LIN {X 0,Y 92.351,Z 360.428,A -85,B 0,C 180,E1 -26835.446,E2 -26835.446} C_VEL
LIN {X 0,Y 91.502,Z 354.022,A -85,B 0,C 180,E1 -26842.823,E2 -26842.823} C_VEL
LIN {X 0,Y 91.802,Z 346.376,A -85,B 0,C 180,E1 -26849.841,E2 -26849.841} C_VEL
LIN {X 0,Y 92.482,Z 339.735,A -85,B 0,C 180,E1 -26854.849,E2 -26854.849} C_VEL
LIN {X 0,Y 93.803,Z 330.262,A -85,B 0,C 180,E1 -26860.681,E2 -26860.681} C_VEL
LIN {X 0,Y 95.598,Z 319.88,A -85,B 0,C 180,E1 -26865.787,E2 -26865.787} C_VEL
LIN {X 0,Y 97.517,Z 309.227,A -85,B 0,C 180,E1 -26869.896,E2 -26869.896} C_VEL
LIN {X 0,Y 99.765,Z 296.448,A -85,B 0,C 180,E1 -26873.677,E2 -26873.677} C_VEL
LIN {X 0,Y 101.625,Z 284.174,A -85,B 0,C 180,E1 -26876.408,E2 -26876.408} C_VEL
LIN {X 0,Y 103.341,Z 270.11,A -85,B 0,C 180,E1 -26878.615,E2 -26878.615} C_VEL
LIN {X 0,Y 107.967,Z 215.614,A -85,B 0,C 180,E1 -26883.951,E2 -26883.951} C_VEL
LIN {X 0,Y 101.224,Z 196.122,A -85,B 0,C 180,E1 -26887.415,E2 -26887.415} C_VEL
LIN {X 0,Y 94.785,Z 179.575,A -85,B 0,C 180,E1 -26890.931,E2 -26890.931} C_VEL
LIN {X 0,Y 93.797,Z 176.802,A -85,B 0,C 180,E1 -26891.572,E2 -26891.572} C_VEL
LIN {X 0,Y 94.063,Z 176.761,A -85,B 0,C 180,E1 -26897.046,E2 -26897.046} C_VEL
LIN {X 0,Y 94.193,Z 176.751,A -85,B 0,C 180,E1 -26901.416,E2 -26901.416} C_VEL
LIN {X 0,Y 94.794,Z 176.676,A -85,B 0,C 180,E1 -26909.998,E2 -26909.998} C_VEL
LIN {X 0,Y 94.198,Z 176.75,A -85,B 0,C 180,E1 -26918.58,E2 -26918.58} C_VEL
LIN {X 0,Y 94.04,Z 176.769,A -85,B 0,C 180,E1 -26923.708,E2 -26923.708} C_VEL
LIN {X 0,Y 93.691,Z 176.812,A -85,B 0,C 180,E1 -26932.027,E2 -26932.027} C_VEL
LIN {X 0,Y 93.619,Z 176.818,A -85,B 0,C 180,E1 -26936.769,E2 -26936.769} C_VEL
LIN {X 0,Y 93.61,Z 176.821,A -85,B 0,C 180,E1 -26944.328,E2 -26944.328} C_VEL
LIN {X 0,Y 93.63,Z 176.819,A -85,B 0,C 180,E1 -26952.495,E2 -26952.495} C_VEL
LIN {X 0,Y 93.626,Z 176.822,A -85,B 0,C 180,E1 -26958.644,E2 -26958.644} C_VEL
LIN {X 0,Y 93.611,Z 176.824,A -85,B 0,C 180,E1 -26965.671,E2 -26965.671} C_VEL
LIN {X 0,Y 93.666,Z 176.817,A -85,B 0,C 180,E1 -26974.205,E2 -26974.205} C_VEL
LIN {X 0,Y 93.691,Z 176.809,A -85,B 0,C 180,E1 -26977.974,E2 -26977.974} C_VEL
LIN {X 0,Y 94.089,Z 176.758,A -85,B 0,C 180,E1 -26987.053,E2 -26987.053} C_VEL
LIN {X 0,Y 94.198,Z 176.752,A -85,B 0,C 180,E1 -26991.42,E2 -26991.42} C_VEL
LIN {X 0,Y 94.794,Z 176.677,A -85,B 0,C 180,E1 -27000.002,E2 -27000.002} C_VEL
LIN {X 0,Y 94.21,Z 176.751,A -85,B 0,C 180,E1 -27008.582,E2 -27008.582} C_VEL
LIN {X 0,Y 94.034,Z 176.767,A -85,B 0,C 180,E1 -27013.693,E2 -27013.693} C_VEL
LIN {X 0,Y 93.692,Z 176.809,A -85,B 0,C 180,E1 -27022.03,E2 -27022.03} C_VEL
LIN {X 0,Y 93.62,Z 176.821,A -85,B 0,C 180,E1 -27026.772,E2 -27026.772} C_VEL
LIN {X 0,Y 93.599,Z 176.825,A -85,B 0,C 180,E1 -27034.318,E2 -27034.318} C_VEL
LIN {X 0,Y 93.641,Z 176.821,A -85,B 0,C 180,E1 -27042.076,E2 -27042.076} C_VEL
LIN {X 0,Y 94.743,Z 179.831,A -85,B 0,C 180,E1 -27042.784,E2 -27042.784} C_VEL
LIN {X 0,Y 98.916,Z 190.263,A -85,B 0,C 180,E1 -27045.097,E2 -27045.097} C_VEL
LIN {X 0,Y 105.331,Z 213.345,A -85,B 0,C 180,E1 -27049.033,E2 -27049.033} C_VEL
LIN {X 0,Y 106.725,Z 240.471,A -85,B 0,C 180,E1 -27052.191,E2 -27052.191} C_VEL
LIN {X 0,Y 103.42,Z 281.466,A -85,B 0,C 180,E1 -27056.341,E2 -27056.341} C_VEL
LIN {X 0,Y 101.758,Z 295.159,A -85,B 0,C 180,E1 -27058.514,E2 -27058.514} C_VEL
LIN {X 0,Y 99.924,Z 306.73,A -85,B 0,C 180,E1 -27061.085,E2 -27061.085} C_VEL
LIN {X 0,Y 97.629,Z 319.739,A -85,B 0,C 180,E1 -27064.982,E2 -27064.982} C_VEL
LIN {X 0,Y 95.507,Z 331.213,A -85,B 0,C 180,E1 -27069.543,E2 -27069.543} C_VEL
LIN {X 0,Y 94.096,Z 341.62,A -85,B 0,C 180,E1 -27074.848,E2 -27074.848} C_VEL
LIN {X 0,Y 93.264,Z 350.336,A -85,B 0,C 180,E1 -27080.438,E2 -27080.438} C_VEL
LIN {X 0,Y 93.204,Z 358.171,A -85,B 0,C 180,E1 -27086.76,E2 -27086.76} C_VEL
LIN {X 0,Y 93.403,Z 363.548,A -85,B 0,C 180,E1 -27092.158,E2 -27092.158} C_VEL
LIN {X 0,Y 92.94,Z 368.337,A -85,B 0,C 180,E1 -27098.7,E2 -27098.7} C_VEL
LIN {X 0,Y 93.452,Z 372.063,A -85,B 0,C 180,E1 -27105.263,E2 -27105.263} C_VEL
LIN {X 0,Y 95.199,Z 374.914,A -85,B 0,C 180,E1 -27111.663,E2 -27111.663} C_VEL
LIN {X 0,Y 99.586,Z 377.581,A -85,B 0,C 180,E1 -27119.606,E2 -27119.606} C_VEL
LIN {X 0,Y 106.025,Z 378.958,A -85,B 0,C 180,E1 -27126.627,E2 -27126.627} C_VEL
LIN {X 0,Y 114.018,Z 379.091,A -85,B 0,C 180,E1 -27132.692,E2 -27132.692} C_VEL
LIN {X 0,Y 123.472,Z 377.959,A -85,B 0,C 180,E1 -27137.729,E2 -27137.729} C_VEL
LIN {X 0,Y 134.03,Z 375.524,A -85,B 0,C 180,E1 -27141.865,E2 -27141.865} C_VEL
LIN {X 0,Y 145.317,Z 371.768,A -85,B 0,C 180,E1 -27145.305,E2 -27145.305} C_VEL
LIN {X 0,Y 154.3,Z 367.94,A -85,B 0,C 180,E1 -27147.421,E2 -27147.421} C_VEL
LIN {X 0,Y 160.353,Z 364.917,A -85,B 0,C 180,E1 -27148.639,E2 -27148.639} C_VEL
LIN {X 0,Y 160.723,Z 364.637,A -85,B 0,C 180,E1 -27149.394,E2 -27149.394} C_VEL
LIN {X 0,Y 149.736,Z 369.187,A -85,B 0,C 180,E1 -27152.006,E2 -27152.006} C_VEL
LIN {X 0,Y 139.588,Z 372.252,A -85,B 0,C 180,E1 -27154.996,E2 -27154.996} C_VEL
LIN {X 0,Y 137.751,Z 372.695,A -85,B 0,C 180,E1 -27155.614,E2 -27155.614} C_VEL
LIN {X 0,Y 132.899,Z 373.732,A -85,B 0,C 180,E1 -27156.983,E2 -27156.983} C_VEL
LIN {X 0,Y 123.979,Z 374.999,A -85,B 0,C 180,E1 -27158.851,E2 -27158.851} C_VEL
LIN {X 0,Y 115.232,Z 375.421,A -85,B 0,C 180,E1 -27161.053,E2 -27161.053} C_VEL
LIN {X 0,Y 110.768,Z 375.21,A -85,B 0,C 180,E1 -27162.998,E2 -27162.998} C_VEL
LIN {X 0,Y 103.035,Z 373.937,A -85,B 0,C 180,E1 -27168.191,E2 -27168.191} C_VEL
LIN {X 0,Y 98.79,Z 372.63,A -85,B 0,C 180,E1 -27171.819,E2 -27171.819} C_VEL
LIN {X 0,Y 93.327,Z 369.871,A -85,B 0,C 180,E1 -27177.841,E2 -27177.841} C_VEL
LIN {X 0,Y 89.087,Z 366.169,A -85,B 0,C 180,E1 -27184.523,E2 -27184.523} C_VEL
LIN {X 0,Y 86.188,Z 361.281,A -85,B 0,C 180,E1 -27191.892,E2 -27191.892} C_VEL
LIN {X 0,Y 84.732,Z 355.371,A -85,B 0,C 180,E1 -27199.375,E2 -27199.375} C_VEL
LIN {X 0,Y 84.582,Z 349.274,A -85,B 0,C 180,E1 -27205.861,E2 -27205.861} C_VEL
LIN {X 0,Y 85.129,Z 342.003,A -85,B 0,C 180,E1 -27212.225,E2 -27212.225} C_VEL
LIN {X 0,Y 86.35,Z 332.15,A -85,B 0,C 180,E1 -27219.105,E2 -27219.105} C_VEL
LIN {X 0,Y 88.2,Z 321.243,A -85,B 0,C 180,E1 -27225.064,E2 -27225.064} C_VEL
LIN {X 0,Y 90.086,Z 310.909,A -85,B 0,C 180,E1 -27229.518,E2 -27229.518} C_VEL
LIN {X 0,Y 92.208,Z 299.417,A -85,B 0,C 180,E1 -27233.381,E2 -27233.381} C_VEL
LIN {X 0,Y 94.384,Z 285.776,A -85,B 0,C 180,E1 -27236.815,E2 -27236.815} C_VEL
LIN {X 0,Y 96.163,Z 272.766,A -85,B 0,C 180,E1 -27239.129,E2 -27239.129} C_VEL
LIN {X 0,Y 98.117,Z 251.11,A -85,B 0,C 180,E1 -27241.602,E2 -27241.602} C_VEL
LIN {X 0,Y 101.067,Z 216.668,A -85,B 0,C 180,E1 -27245.079,E2 -27245.079} C_VEL
LIN {X 0,Y 93.632,Z 195.122,A -85,B 0,C 180,E1 -27249.255,E2 -27249.255} C_VEL
LIN {X 0,Y 87.72,Z 180.438,A -85,B 0,C 180,E1 -27252.769,E2 -27252.769} C_VEL
LIN {X 0,Y 86.787,Z 177.673,A -85,B 0,C 180,E1 -27253.533,E2 -27253.533} C_VEL
LIN {X 0,Y 87.097,Z 177.636,A -85,B 0,C 180,E1 -27260.711,E2 -27260.711} C_VEL
LIN {X 0,Y 87.721,Z 177.557,A -85,B 0,C 180,E1 -27269.998,E2 -27269.998} C_VEL
LIN {X 0,Y 87.106,Z 177.632,A -85,B 0,C 180,E1 -27279.284,E2 -27279.284} C_VEL
LIN {X 0,Y 86.948,Z 177.653,A -85,B 0,C 180,E1 -27284.086,E2 -27284.086} C_VEL
LIN {X 0,Y 86.584,Z 177.7,A -85,B 0,C 180,E1 -27293.942,E2 -27293.942} C_VEL
LIN {X 0,Y 86.475,Z 177.709,A -85,B 0,C 180,E1 -27299.183,E2 -27299.183} C_VEL
LIN {X 0,Y 86.535,Z 177.699,A -85,B 0,C 180,E1 -27305.695,E2 -27305.695} C_VEL
LIN {X 0,Y 86.557,Z 177.698,A -85,B 0,C 180,E1 -27313.053,E2 -27313.053} C_VEL
LIN {X 0,Y 86.55,Z 177.704,A -85,B 0,C 180,E1 -27319.49,E2 -27319.49} C_VEL
LIN {X 0,Y 86.559,Z 177.701,A -85,B 0,C 180,E1 -27325.367,E2 -27325.367} C_VEL
LIN {X 0,Y 86.583,Z 177.697,A -85,B 0,C 180,E1 -27333.233,E2 -27333.233} C_VEL
LIN {X 0,Y 86.645,Z 177.688,A -85,B 0,C 180,E1 -27341.07,E2 -27341.07} C_VEL
LIN {X 0,Y 86.967,Z 177.648,A -85,B 0,C 180,E1 -27345.971,E2 -27345.971} C_VEL
LIN {X 0,Y 87.106,Z 177.634,A -85,B 0,C 180,E1 -27350.716,E2 -27350.716} C_VEL
LIN {X 0,Y 87.721,Z 177.558,A -85,B 0,C 180,E1 -27360.002,E2 -27360.002} C_VEL
LIN {X 0,Y 87.114,Z 177.633,A -85,B 0,C 180,E1 -27369.287,E2 -27369.287} C_VEL
LIN {X 0,Y 86.949,Z 177.65,A -85,B 0,C 180,E1 -27374.089,E2 -27374.089} C_VEL
LIN {X 0,Y 86.586,Z 177.699,A -85,B 0,C 180,E1 -27383.946,E2 -27383.946} C_VEL
LIN {X 0,Y 86.475,Z 177.705,A -85,B 0,C 180,E1 -27389.187,E2 -27389.187} C_VEL
LIN {X 0,Y 86.521,Z 177.703,A -85,B 0,C 180,E1 -27395.683,E2 -27395.683} C_VEL
LIN {X 0,Y 86.529,Z 177.852,A -85,B 0,C 180,E1 -27400.186,E2 -27400.186} C_VEL
LIN {X 0,Y 88.646,Z 183.012,A -85,B 0,C 180,E1 -27401.528,E2 -27401.528} C_VEL
LIN {X 0,Y 92.717,Z 193.174,A -85,B 0,C 180,E1 -27403.954,E2 -27403.954} C_VEL
LIN {X 0,Y 98.684,Z 215.03,A -85,B 0,C 180,E1 -27407.971,E2 -27407.971} C_VEL
LIN {X 0,Y 99.874,Z 240.558,A -85,B 0,C 180,E1 -27411.166,E2 -27411.166} C_VEL
LIN {X 0,Y 96.441,Z 281.612,A -85,B 0,C 180,E1 -27415.616,E2 -27415.616} C_VEL
LIN {X 0,Y 94.812,Z 294.504,A -85,B 0,C 180,E1 -27417.808,E2 -27417.808} C_VEL
LIN {X 0,Y 92.919,Z 306.132,A -85,B 0,C 180,E1 -27420.554,E2 -27420.554} C_VEL
LIN {X 0,Y 90.555,Z 319.15,A -85,B 0,C 180,E1 -27424.734,E2 -27424.734} C_VEL
LIN {X 0,Y 88.426,Z 330.571,A -85,B 0,C 180,E1 -27429.654,E2 -27429.654} C_VEL
LIN {X 0,Y 87.135,Z 340.166,A -85,B 0,C 180,E1 -27434.926,E2 -27434.926} C_VEL
LIN {X 0,Y 86.384,Z 348.549,A -85,B 0,C 180,E1 -27440.637,E2 -27440.637} C_VEL
LIN {X 0,Y 86.382,Z 356.895,A -85,B 0,C 180,E1 -27447.67,E2 -27447.67} C_VEL
LIN {X 0,Y 86.603,Z 361.336,A -85,B 0,C 180,E1 -27452.327,E2 -27452.327} C_VEL
LIN {X 0,Y 86.258,Z 364.886,A -85,B 0,C 180,E1 -27457.022,E2 -27457.022} C_VEL
LIN {X 0,Y 86.463,Z 369.143,A -85,B 0,C 180,E1 -27464.116,E2 -27464.116} C_VEL
LIN {X 0,Y 88.757,Z 373.493,A -85,B 0,C 180,E1 -27473.325,E2 -27473.325} C_VEL
LIN {X 0,Y 93.53,Z 376.466,A -85,B 0,C 180,E1 -27481.737,E2 -27481.737} C_VEL
LIN {X 0,Y 100.426,Z 378.161,A -85,B 0,C 180,E1 -27489.04,E2 -27489.04} C_VEL
LIN {X 0,Y 108.92,Z 378.615,A -85,B 0,C 180,E1 -27495.218,E2 -27495.218} C_VEL
LIN {X 0,Y 118.822,Z 377.86,A -85,B 0,C 180,E1 -27500.258,E2 -27500.258} C_VEL
LIN {X 0,Y 129.784,Z 375.856,A -85,B 0,C 180,E1 -27504.32,E2 -27504.32} C_VEL
LIN {X 0,Y 141.416,Z 372.548,A -85,B 0,C 180,E1 -27507.658,E2 -27507.658} C_VEL
LIN {X 0,Y 147.52,Z 370.327,A -85,B 0,C 180,E1 -27509.043,E2 -27509.043} C_VEL
LIN {X 0,Y 146.705,Z 370.553,A -85,B 0,C 180,E1 -27509.578,E2 -27509.578} C_VEL
LIN {X 0,Y 133.944,Z 373.781,A -85,B 0,C 180,E1 -27513.126,E2 -27513.126} C_VEL
LIN {X 0,Y 121.594,Z 375.353,A -85,B 0,C 180,E1 -27517.638,E2 -27517.638} C_VEL
LIN {X 0,Y 110.768,Z 375.21,A -85,B 0,C 180,E1 -27522.998,E2 -27522.998} C_VEL
LIN {X 0,Y 106.467,Z 374.769,A -85,B 0,C 180,E1 -27525.123,E2 -27525.123} C_VEL
LIN {X 0,Y 98.494,Z 373.407,A -85,B 0,C 180,E1 -27528.331,E2 -27528.331} C_VEL
LIN {X 0,Y 91.021,Z 371.275,A -85,B 0,C 180,E1 -27532.057,E2 -27532.057} C_VEL
LIN {X 0,Y 87.655,Z 369.634,A -85,B 0,C 180,E1 -27535.004,E2 -27535.004} C_VEL
LIN {X 0,Y 82.729,Z 365.476,A -85,B 0,C 180,E1 -27542.433,E2 -27542.433} C_VEL
LIN {X 0,Y 79.044,Z 359.168,A -85,B 0,C 180,E1 -27552.021,E2 -27552.021} C_VEL
LIN {X 0,Y 77.691,Z 351.807,A -85,B 0,C 180,E1 -27561.212,E2 -27561.212} C_VEL
LIN {X 0,Y 77.776,Z 344.892,A -85,B 0,C 180,E1 -27568.318,E2 -27568.318} C_VEL
LIN {X 0,Y 78.474,Z 337.481,A -85,B 0,C 180,E1 -27574.618,E2 -27574.618} C_VEL
LIN {X 0,Y 79.851,Z 327.7,A -85,B 0,C 180,E1 -27581.305,E2 -27581.305} C_VEL
LIN {X 0,Y 81.805,Z 316.889,A -85,B 0,C 180,E1 -27587.09,E2 -27587.09} C_VEL
LIN {X 0,Y 83.908,Z 305.754,A -85,B 0,C 180,E1 -27591.74,E2 -27591.74} C_VEL
LIN {X 0,Y 86.18,Z 293.338,A -85,B 0,C 180,E1 -27595.656,E2 -27595.656} C_VEL
LIN {X 0,Y 88.299,Z 279.63,A -85,B 0,C 180,E1 -27598.825,E2 -27598.825} C_VEL
LIN {X 0,Y 89.719,Z 267.085,A -85,B 0,C 180,E1 -27600.824,E2 -27600.824} C_VEL
LIN {X 0,Y 94.234,Z 217.928,A -85,B 0,C 180,E1 -27606.271,E2 -27606.271} C_VEL
LIN {X 0,Y 87.202,Z 197.474,A -85,B 0,C 180,E1 -27610.578,E2 -27610.578} C_VEL
LIN {X 0,Y 81.948,Z 184.113,A -85,B 0,C 180,E1 -27614.054,E2 -27614.054} C_VEL
LIN {X 0,Y 79.877,Z 178.778,A -85,B 0,C 180,E1 -27615.579,E2 -27615.579} C_VEL
LIN {X 0,Y 79.865,Z 178.529,A -85,B 0,C 180,E1 -27615.871,E2 -27615.871} C_VEL
LIN {X 0,Y 79.976,Z 178.523,A -85,B 0,C 180,E1 -27619.876,E2 -27619.876} C_VEL
LIN {X 0,Y 80.649,Z 178.439,A -85,B 0,C 180,E1 -27629.998,E2 -27629.998} C_VEL
LIN {X 0,Y 79.991,Z 178.515,A -85,B 0,C 180,E1 -27640.119,E2 -27640.119} C_VEL
LIN {X 0,Y 79.76,Z 178.55,A -85,B 0,C 180,E1 -27645.326,E2 -27645.326} C_VEL
LIN {X 0,Y 79.511,Z 178.574,A -85,B 0,C 180,E1 -27650.703,E2 -27650.703} C_VEL
LIN {X 0,Y 79.48,Z 178.577,A -85,B 0,C 180,E1 -27657.845,E2 -27657.845} C_VEL
LIN {X 0,Y 79.449,Z 178.583,A -85,B 0,C 180,E1 -27667.241,E2 -27667.241} C_VEL
LIN {X 0,Y 79.464,Z 178.579,A -85,B 0,C 180,E1 -27675.032,E2 -27675.032} C_VEL
LIN {X 0,Y 79.45,Z 178.58,A -85,B 0,C 180,E1 -27682.758,E2 -27682.758} C_VEL
LIN {X 0,Y 79.482,Z 178.579,A -85,B 0,C 180,E1 -27692.153,E2 -27692.153} C_VEL
LIN {X 0,Y 79.512,Z 178.573,A -85,B 0,C 180,E1 -27699.297,E2 -27699.297} C_VEL
LIN {X 0,Y 79.839,Z 178.537,A -85,B 0,C 180,E1 -27705.527,E2 -27705.527} C_VEL
LIN {X 0,Y 79.991,Z 178.519,A -85,B 0,C 180,E1 -27709.881,E2 -27709.881} C_VEL
LIN {X 0,Y 80.649,Z 178.439,A -85,B 0,C 180,E1 -27720.002,E2 -27720.002} C_VEL
LIN {X 0,Y 79.993,Z 178.518,A -85,B 0,C 180,E1 -27730.122,E2 -27730.122} C_VEL
LIN {X 0,Y 79.761,Z 178.549,A -85,B 0,C 180,E1 -27735.33,E2 -27735.33} C_VEL
LIN {X 0,Y 79.513,Z 178.573,A -85,B 0,C 180,E1 -27740.707,E2 -27740.707} C_VEL
LIN {X 0,Y 79.481,Z 178.578,A -85,B 0,C 180,E1 -27747.847,E2 -27747.847} C_VEL
LIN {X 0,Y 79.443,Z 178.581,A -85,B 0,C 180,E1 -27757.235,E2 -27757.235} C_VEL
LIN {X 0,Y 79.44,Z 178.582,A -85,B 0,C 180,E1 -27757.878,E2 -27757.878} C_VEL
LIN {X 0,Y 80.432,Z 181.432,A -85,B 0,C 180,E1 -27758.708,E2 -27758.708} C_VEL
LIN {X 0,Y 85.393,Z 192.723,A -85,B 0,C 180,E1 -27761.942,E2 -27761.942} C_VEL
LIN {X 0,Y 89.063,Z 205.266,A -85,B 0,C 180,E1 -27764.626,E2 -27764.626} C_VEL
LIN {X 0,Y 92.048,Z 217.164,A -85,B 0,C 180,E1 -27766.835,E2 -27766.835} C_VEL
LIN {X 0,Y 93.078,Z 240.438,A -85,B 0,C 180,E1 -27769.967,E2 -27769.967} C_VEL
LIN {X 0,Y 89.562,Z 280.628,A -85,B 0,C 180,E1 -27774.641,E2 -27774.641} C_VEL
LIN {X 0,Y 87.906,Z 293.587,A -85,B 0,C 180,E1 -27777.001,E2 -27777.001} C_VEL
LIN {X 0,Y 85.956,Z 305.243,A -85,B 0,C 180,E1 -27779.949,E2 -27779.949} C_VEL
LIN {X 0,Y 83.546,Z 318.246,A -85,B 0,C 180,E1 -27784.463,E2 -27784.463} C_VEL
LIN {X 0,Y 81.385,Z 329.761,A -85,B 0,C 180,E1 -27789.795,E2 -27789.795} C_VEL
LIN {X 0,Y 79.98,Z 340.754,A -85,B 0,C 180,E1 -27796.433,E2 -27796.433} C_VEL
LIN {X 0,Y 79.417,Z 348.596,A -85,B 0,C 180,E1 -27802.374,E2 -27802.374} C_VEL
LIN {X 0,Y 79.585,Z 355.553,A -85,B 0,C 180,E1 -27808.737,E2 -27808.737} C_VEL
LIN {X 0,Y 79.808,Z 359.014,A -85,B 0,C 180,E1 -27812.525,E2 -27812.525} C_VEL
LIN {X 0,Y 79.568,Z 362.74,A -85,B 0,C 180,E1 -27817.615,E2 -27817.615} C_VEL
LIN {X 0,Y 80.239,Z 368.574,A -85,B 0,C 180,E1 -27827.854,E2 -27827.854} C_VEL
LIN {X 0,Y 82.417,Z 371.927,A -85,B 0,C 180,E1 -27835.239,E2 -27835.239} C_VEL
LIN {X 0,Y 87.664,Z 375.208,A -85,B 0,C 180,E1 -27844.14,E2 -27844.14} C_VEL
LIN {X 0,Y 95.053,Z 377.24,A -85,B 0,C 180,E1 -27851.718,E2 -27851.718} C_VEL
LIN {X 0,Y 104.064,Z 378.056,A -85,B 0,C 180,E1 -27857.98,E2 -27857.98} C_VEL
LIN {X 0,Y 114.428,Z 377.687,A -85,B 0,C 180,E1 -27862.984,E2 -27862.984} C_VEL
LIN {X 0,Y 125.782,Z 376.089,A -85,B 0,C 180,E1 -27866.944,E2 -27866.944} C_VEL
LIN {X 0,Y 131.672,Z 374.799,A -85,B 0,C 180,E1 -27868.651,E2 -27868.651} C_VEL
LIN {X 0,Y 133.177,Z 374.323,A -85,B 0,C 180,E1 -27869.701,E2 -27869.701} C_VEL
LIN {X 0,Y 123.077,Z 375.674,A -85,B 0,C 180,E1 -27872.817,E2 -27872.817} C_VEL
LIN {X 0,Y 115.793,Z 376.028,A -85,B 0,C 180,E1 -27875.567,E2 -27875.567} C_VEL
LIN {X 0,Y 105.417,Z 375.414,A -85,B 0,C 180,E1 -27880.527,E2 -27880.527} C_VEL
LIN {X 0,Y 95.489,Z 373.242,A -85,B 0,C 180,E1 -27887.242,E2 -27887.242} C_VEL
LIN {X 0,Y 89.18,Z 370.55,A -85,B 0,C 180,E1 -27893.209,E2 -27893.209} C_VEL
LIN {X 0,Y 87.655,Z 369.634,A -85,B 0,C 180,E1 -27895.004,E2 -27895.004} C_VEL
LIN {X 0,Y 84.598,Z 367.791,A -85,B 0,C 180,E1 -27898.135,E2 -27898.135} C_VEL
LIN {X 0,Y 78.699,Z 364.017,A -85,B 0,C 180,E1 -27903.064,E2 -27903.064} C_VEL
LIN {X 0,Y 73.582,Z 359.497,A -85,B 0,C 180,E1 -27908.531,E2 -27908.531} C_VEL
LIN {X 0,Y 71.904,Z 356.563,A -85,B 0,C 180,E1 -27912.38,E2 -27912.38} C_VEL
LIN {X 0,Y 70.76,Z 349.115,A -85,B 0,C 180,E1 -27921.865,E2 -27921.865} C_VEL
LIN {X 0,Y 71.017,Z 341.606,A -85,B 0,C 180,E1 -27929.655,E2 -27929.655} C_VEL
LIN {X 0,Y 71.958,Z 332.755,A -85,B 0,C 180,E1 -27937.081,E2 -27937.081} C_VEL
LIN {X 0,Y 73.55,Z 322.642,A -85,B 0,C 180,E1 -27943.847,E2 -27943.847} C_VEL
LIN {X 0,Y 75.73,Z 311.186,A -85,B 0,C 180,E1 -27949.834,E2 -27949.834} C_VEL
LIN {X 0,Y 77.906,Z 299.975,A -85,B 0,C 180,E1 -27954.278,E2 -27954.278} C_VEL
LIN {X 0,Y 80.336,Z 286.072,A -85,B 0,C 180,E1 -27958.336,E2 -27958.336} C_VEL
LIN {X 0,Y 82.359,Z 271.903,A -85,B 0,C 180,E1 -27961.16,E2 -27961.16} C_VEL
LIN {X 0,Y 86.345,Z 230.389,A -85,B 0,C 180,E1 -27966.296,E2 -27966.296} C_VEL
LIN {X 0,Y 87.453,Z 219.393,A -85,B 0,C 180,E1 -27967.533,E2 -27967.533} C_VEL
LIN {X 0,Y 81.166,Z 200.697,A -85,B 0,C 180,E1 -27971.868,E2 -27971.868} C_VEL
LIN {X 0,Y 76.043,Z 187.435,A -85,B 0,C 180,E1 -27975.606,E2 -27975.606} C_VEL
LIN {X 0,Y 72.922,Z 179.748,A -85,B 0,C 180,E1 -27978.112,E2 -27978.112} C_VEL
LIN {X 0,Y 72.865,Z 179.406,A -85,B 0,C 180,E1 -27978.489,E2 -27978.489} C_VEL
LIN {X 0,Y 73.575,Z 179.32,A -85,B 0,C 180,E1 -27989.998,E2 -27989.998} C_VEL
LIN {X 0,Y 72.878,Z 179.399,A -85,B 0,C 180,E1 -28001.118,E2 -28001.118} C_VEL
LIN {X 0,Y 72.58,Z 179.443,A -85,B 0,C 180,E1 -28006.885,E2 -28006.885} C_VEL
LIN {X 0,Y 72.391,Z 179.468,A -85,B 0,C 180,E1 -28012.849,E2 -28012.849} C_VEL
LIN {X 0,Y 72.373,Z 179.464,A -85,B 0,C 180,E1 -28019.081,E2 -28019.081} C_VEL
LIN {X 0,Y 72.335,Z 179.467,A -85,B 0,C 180,E1 -28025.656,E2 -28025.656} C_VEL
LIN {X 0,Y 72.31,Z 179.473,A -85,B 0,C 180,E1 -28032.868,E2 -28032.868} C_VEL
LIN {X 0,Y 72.357,Z 179.467,A -85,B 0,C 180,E1 -28040.987,E2 -28040.987} C_VEL
LIN {X 0,Y 72.336,Z 179.47,A -85,B 0,C 180,E1 -28044.344,E2 -28044.344} C_VEL
LIN {X 0,Y 72.389,Z 179.46,A -85,B 0,C 180,E1 -28050.961,E2 -28050.961} C_VEL
LIN {X 0,Y 72.392,Z 179.464,A -85,B 0,C 180,E1 -28057.152,E2 -28057.152} C_VEL
LIN {X 0,Y 72.733,Z 179.423,A -85,B 0,C 180,E1 -28065.068,E2 -28065.068} C_VEL
LIN {X 0,Y 72.878,Z 179.401,A -85,B 0,C 180,E1 -28068.882,E2 -28068.882} C_VEL
LIN {X 0,Y 73.575,Z 179.32,A -85,B 0,C 180,E1 -28080.002,E2 -28080.002} C_VEL
LIN {X 0,Y 72.878,Z 179.401,A -85,B 0,C 180,E1 -28091.122,E2 -28091.122} C_VEL
LIN {X 0,Y 72.581,Z 179.444,A -85,B 0,C 180,E1 -28096.889,E2 -28096.889} C_VEL
LIN {X 0,Y 72.393,Z 179.464,A -85,B 0,C 180,E1 -28102.853,E2 -28102.853} C_VEL
LIN {X 0,Y 72.376,Z 179.461,A -85,B 0,C 180,E1 -28109.085,E2 -28109.085} C_VEL
LIN {X 0,Y 72.306,Z 179.475,A -85,B 0,C 180,E1 -28115.25,E2 -28115.25} C_VEL
LIN {X 0,Y 73.4,Z 182.395,A -85,B 0,C 180,E1 -28116.217,E2 -28116.217} C_VEL
LIN {X 0,Y 78.274,Z 193.22,A -85,B 0,C 180,E1 -28119.774,E2 -28119.774} C_VEL
LIN {X 0,Y 80.557,Z 199.631,A -85,B 0,C 180,E1 -28121.493,E2 -28121.493} C_VEL
LIN {X 0,Y 85.327,Z 218.12,A -85,B 0,C 180,E1 -28125.462,E2 -28125.462} C_VEL
LIN {X 0,Y 86.228,Z 240.55,A -85,B 0,C 180,E1 -28128.73,E2 -28128.73} C_VEL
LIN {X 0,Y 82.567,Z 280.829,A -85,B 0,C 180,E1 -28133.809,E2 -28133.809} C_VEL
LIN {X 0,Y 80.846,Z 293.597,A -85,B 0,C 180,E1 -28136.348,E2 -28136.348} C_VEL
LIN {X 0,Y 78.654,Z 305.996,A -85,B 0,C 180,E1 -28139.829,E2 -28139.829} C_VEL
LIN {X 0,Y 76.542,Z 317.338,A -85,B 0,C 180,E1 -28144.144,E2 -28144.144} C_VEL
LIN {X 0,Y 74.337,Z 328.947,A -85,B 0,C 180,E1 -28149.962,E2 -28149.962} C_VEL
LIN {X 0,Y 73.023,Z 339.669,A -85,B 0,C 180,E1 -28157.015,E2 -28157.015} C_VEL
LIN {X 0,Y 72.564,Z 348.536,A -85,B 0,C 180,E1 -28164.444,E2 -28164.444} C_VEL
LIN {X 0,Y 72.962,Z 355.297,A -85,B 0,C 180,E1 -28171.382,E2 -28171.382} C_VEL
LIN {X 0,Y 73.103,Z 358.606,A -85,B 0,C 180,E1 -28175.519,E2 -28175.519} C_VEL
LIN {X 0,Y 72.934,Z 363.505,A -85,B 0,C 180,E1 -28183.459,E2 -28183.459} C_VEL
LIN {X 0,Y 74.405,Z 367.92,A -85,B 0,C 180,E1 -28192.201,E2 -28192.201} C_VEL
LIN {X 0,Y 78.79,Z 372.206,A -85,B 0,C 180,E1 -28202.359,E2 -28202.359} C_VEL
LIN {X 0,Y 85.711,Z 375.195,A -85,B 0,C 180,E1 -28210.996,E2 -28210.996} C_VEL
LIN {X 0,Y 94.509,Z 376.966,A -85,B 0,C 180,E1 -28218.044,E2 -28218.044} C_VEL
LIN {X 0,Y 104.738,Z 377.54,A -85,B 0,C 180,E1 -28223.633,E2 -28223.633} C_VEL
LIN {X 0,Y 116.085,Z 376.929,A -85,B 0,C 180,E1 -28227.953,E2 -28227.953} C_VEL
LIN {X 0,Y 118.009,Z 376.707,A -85,B 0,C 180,E1 -28228.548,E2 -28228.548} C_VEL
LIN {X 0,Y 119.865,Z 376.399,A -85,B 0,C 180,E1 -28229.828,E2 -28229.828} C_VEL
LIN {X 0,Y 109.849,Z 376.469,A -85,B 0,C 180,E1 -28233.393,E2 -28233.393} C_VEL
LIN {X 0,Y 98.131,Z 375.095,A -85,B 0,C 180,E1 -28239.015,E2 -28239.015} C_VEL
LIN {X 0,Y 87.951,Z 372.179,A -85,B 0,C 180,E1 -28246.128,E2 -28246.128} C_VEL
LIN {X 0,Y 79.723,Z 367.624,A -85,B 0,C 180,E1 -28254.941,E2 -28254.941} C_VEL
LIN {X 0,Y 75.173,Z 363.052,A -85,B 0,C 180,E1 -28262.677,E2 -28262.677} C_VEL
LIN {X 0,Y 71.904,Z 356.563,A -85,B 0,C 180,E1 -28272.38,E2 -28272.38} C_VEL
LIN {X 0,Y 70.592,Z 353.473,A -85,B 0,C 180,E1 -28276.255,E2 -28276.255} C_VEL
LIN {X 0,Y 68.718,Z 350.021,A -85,B 0,C 180,E1 -28279.92,E2 -28279.92} C_VEL
LIN {X 0,Y 65.106,Z 342.359,A -85,B 0,C 180,E1 -28287.233,E2 -28287.233} C_VEL
LIN {X 0,Y 64.351,Z 338.253,A -85,B 0,C 180,E1 -28291.038,E2 -28291.038} C_VEL
LIN {X 0,Y 64.387,Z 336.838,A -85,B 0,C 180,E1 -28292.312,E2 -28292.312} C_VEL
LIN {X 0,Y 65.744,Z 326.301,A -85,B 0,C 180,E1 -28300.873,E2 -28300.873} C_VEL
LIN {X 0,Y 67.713,Z 315.47,A -85,B 0,C 180,E1 -28307.686,E2 -28307.686} C_VEL
LIN {X 0,Y 70.05,Z 303.585,A -85,B 0,C 180,E1 -28313.378,E2 -28313.378} C_VEL
LIN {X 0,Y 72.322,Z 291.896,A -85,B 0,C 180,E1 -28317.585,E2 -28317.585} C_VEL
LIN {X 0,Y 74.66,Z 277.702,A -85,B 0,C 180,E1 -28321.212,E2 -28321.212} C_VEL
LIN {X 0,Y 76.261,Z 263.956,A -85,B 0,C 180,E1 -28323.566,E2 -28323.566} C_VEL
LIN {X 0,Y 80.665,Z 220.64,A -85,B 0,C 180,E1 -28329.06,E2 -28329.06} C_VEL
LIN {X 0,Y 74.815,Z 203.089,A -85,B 0,C 180,E1 -28333.495,E2 -28333.495} C_VEL
LIN {X 0,Y 70.277,Z 190.976,A -85,B 0,C 180,E1 -28337.255,E2 -28337.255} C_VEL
LIN {X 0,Y 66.729,Z 182.984,A -85,B 0,C 180,E1 -28340.335,E2 -28340.335} C_VEL
LIN {X 0,Y 65.823,Z 180.285,A -85,B 0,C 180,E1 -28341.362,E2 -28341.362} C_VEL
LIN {X 0,Y 66.499,Z 180.201,A -85,B 0,C 180,E1 -28349.998,E2 -28349.998} C_VEL
LIN {X 0,Y 65.77,Z 180.285,A -85,B 0,C 180,E1 -28362.338,E2 -28362.338} C_VEL
LIN {X 0,Y 65.382,Z 180.333,A -85,B 0,C 180,E1 -28368.81,E2 -28368.81} C_VEL
LIN {X 0,Y 65.243,Z 180.355,A -85,B 0,C 180,E1 -28375.521,E2 -28375.521} C_VEL
LIN {X 0,Y 65.212,Z 180.362,A -85,B 0,C 180,E1 -28382.603,E2 -28382.603} C_VEL
LIN {X 0,Y 65.247,Z 180.357,A -85,B 0,C 180,E1 -28391.066,E2 -28391.066} C_VEL
LIN {X 0,Y 65.264,Z 180.354,A -85,B 0,C 180,E1 -28399.754,E2 -28399.754} C_VEL
LIN {X 0,Y 65.257,Z 180.351,A -85,B 0,C 180,E1 -28409.49,E2 -28409.49} C_VEL
LIN {X 0,Y 65.245,Z 180.358,A -85,B 0,C 180,E1 -28414.48,E2 -28414.48} C_VEL
LIN {X 0,Y 65.634,Z 180.309,A -85,B 0,C 180,E1 -28424.509,E2 -28424.509} C_VEL
LIN {X 0,Y 65.77,Z 180.284,A -85,B 0,C 180,E1 -28427.662,E2 -28427.662} C_VEL
LIN {X 0,Y 66.499,Z 180.202,A -85,B 0,C 180,E1 -28440.002,E2 -28440.002} C_VEL
LIN {X 0,Y 65.778,Z 180.283,A -85,B 0,C 180,E1 -28452.341,E2 -28452.341} C_VEL
LIN {X 0,Y 65.384,Z 180.336,A -85,B 0,C 180,E1 -28458.814,E2 -28458.814} C_VEL
LIN {X 0,Y 65.238,Z 180.359,A -85,B 0,C 180,E1 -28465.528,E2 -28465.528} C_VEL
LIN {X 0,Y 65.292,Z 180.351,A -85,B 0,C 180,E1 -28472.075,E2 -28472.075} C_VEL
LIN {X 0,Y 66.418,Z 183.431,A -85,B 0,C 180,E1 -28473.294,E2 -28473.294} C_VEL
LIN {X 0,Y 71.516,Z 194.42,A -85,B 0,C 180,E1 -28477.531,E2 -28477.531} C_VEL
LIN {X 0,Y 74.266,Z 201.919,A -85,B 0,C 180,E1 -28479.782,E2 -28479.782} C_VEL
LIN {X 0,Y 78.68,Z 219.568,A -85,B 0,C 180,E1 -28483.934,E2 -28483.934} C_VEL
LIN {X 0,Y 79.422,Z 240.914,A -85,B 0,C 180,E1 -28487.336,E2 -28487.336} C_VEL
LIN {X 0,Y 75.676,Z 280.153,A -85,B 0,C 180,E1 -28492.662,E2 -28492.662} C_VEL
LIN {X 0,Y 73.801,Z 293.612,A -85,B 0,C 180,E1 -28495.571,E2 -28495.571} C_VEL
LIN {X 0,Y 71.37,Z 306.72,A -85,B 0,C 180,E1 -28499.693,E2 -28499.693} C_VEL
LIN {X 0,Y 69.247,Z 317.733,A -85,B 0,C 180,E1 -28504.45,E2 -28504.45} C_VEL
LIN {X 0,Y 67.21,Z 328.731,A -85,B 0,C 180,E1 -28510.692,E2 -28510.692} C_VEL
LIN {X 0,Y 66.11,Z 338.381,A -85,B 0,C 180,E1 -28517.727,E2 -28517.727} C_VEL
LIN {X 0,Y 65.769,Z 346.84,A -85,B 0,C 180,E1 -28525.405,E2 -28525.405} C_VEL
LIN {X 0,Y 66.307,Z 353.782,A -85,B 0,C 180,E1 -28533.04,E2 -28533.04} C_VEL
LIN {X 0,Y 66.462,Z 356.104,A -85,B 0,C 180,E1 -28536.072,E2 -28536.072} C_VEL
LIN {X 0,Y 66.524,Z 361.868,A -85,B 0,C 180,E1 -28545.973,E2 -28545.973} C_VEL
LIN {X 0,Y 69.102,Z 367.227,A -85,B 0,C 180,E1 -28557.239,E2 -28557.239} C_VEL
LIN {X 0,Y 73.044,Z 370.577,A -85,B 0,C 180,E1 -28565.263,E2 -28565.263} C_VEL
LIN {X 0,Y 80.56,Z 373.874,A -85,B 0,C 180,E1 -28574.262,E2 -28574.262} C_VEL
LIN {X 0,Y 89.958,Z 375.97,A -85,B 0,C 180,E1 -28581.378,E2 -28581.378} C_VEL
LIN {X 0,Y 100.707,Z 376.905,A -85,B 0,C 180,E1 -28586.873,E2 -28586.873} C_VEL
LIN {X 0,Y 106.518,Z 376.949,A -85,B 0,C 180,E1 -28589.065,E2 -28589.065} C_VEL
LIN {X 0,Y 104.762,Z 376.712,A -85,B 0,C 180,E1 -28590.707,E2 -28590.707} C_VEL
LIN {X 0,Y 96.729,Z 375.645,A -85,B 0,C 180,E1 -28594.153,E2 -28594.153} C_VEL
LIN {X 0,Y 85.488,Z 372.78,A -85,B 0,C 180,E1 -28600.8,E2 -28600.8} C_VEL
LIN {X 0,Y 78.146,Z 369.508,A -85,B 0,C 180,E1 -28607.095,E2 -28607.095} C_VEL
LIN {X 0,Y 72.195,Z 365.399,A -85,B 0,C 180,E1 -28614.411,E2 -28614.411} C_VEL
LIN {X 0,Y 67.09,Z 359.292,A -85,B 0,C 180,E1 -28624.504,E2 -28624.504} C_VEL
LIN {X 0,Y 64.33,Z 351.422,A -85,B 0,C 180,E1 -28635.844,E2 -28635.844} C_VEL
LIN {X 0,Y 63.899,Z 344.564,A -85,B 0,C 180,E1 -28644.356,E2 -28644.356} C_VEL
LIN {X 0,Y 64.387,Z 336.838,A -85,B 0,C 180,E1 -28652.312,E2 -28652.312} C_VEL
LIN {X 0,Y 64.172,Z 332.601,A -85,B 0,C 180,E1 -28655.902,E2 -28655.902} C_VEL
LIN {X 0,Y 62.385,Z 324.99,A -85,B 0,C 180,E1 -28661.426,E2 -28661.426} C_VEL
LIN {X 0,Y 60.912,Z 316.862,A -85,B 0,C 180,E1 -28666.736,E2 -28666.736} C_VEL
LIN {X 0,Y 61.236,Z 311.795,A -85,B 0,C 180,E1 -28669.719,E2 -28669.719} C_VEL
LIN {X 0,Y 63.701,Z 299.814,A -85,B 0,C 180,E1 -28675.499,E2 -28675.499} C_VEL
LIN {X 0,Y 66.291,Z 286.285,A -85,B 0,C 180,E1 -28680.224,E2 -28680.224} C_VEL
LIN {X 0,Y 68.588,Z 271.36,A -85,B 0,C 180,E1 -28683.707,E2 -28683.707} C_VEL
LIN {X 0,Y 73.816,Z 221.568,A -85,B 0,C 180,E1 -28690.799,E2 -28690.799} C_VEL
LIN {X 0,Y 67.875,Z 203.568,A -85,B 0,C 180,E1 -28695.988,E2 -28695.988} C_VEL
LIN {X 0,Y 62.811,Z 190.132,A -85,B 0,C 180,E1 -28700.942,E2 -28700.942} C_VEL
LIN {X 0,Y 59.071,Z 181.858,A -85,B 0,C 180,E1 -28704.878,E2 -28704.878} C_VEL
LIN {X 0,Y 58.954,Z 181.133,A -85,B 0,C 180,E1 -28705.296,E2 -28705.296} C_VEL
LIN {X 0,Y 59.39,Z 181.086,A -85,B 0,C 180,E1 -28709.997,E2 -28709.997} C_VEL
LIN {X 0,Y 58.816,Z 181.159,A -85,B 0,C 180,E1 -28716.86,E2 -28716.86} C_VEL
LIN {X 0,Y 58.523,Z 181.195,A -85,B 0,C 180,E1 -28726.122,E2 -28726.122} C_VEL
LIN {X 0,Y 58.153,Z 181.234,A -85,B 0,C 180,E1 -28738.906,E2 -28738.906} C_VEL
LIN {X 0,Y 58.072,Z 181.244,A -85,B 0,C 180,E1 -28747.234,E2 -28747.234} C_VEL
LIN {X 0,Y 58.092,Z 181.245,A -85,B 0,C 180,E1 -28756.539,E2 -28756.539} C_VEL
LIN {X 0,Y 58.072,Z 181.242,A -85,B 0,C 180,E1 -28762.766,E2 -28762.766} C_VEL
LIN {X 0,Y 58.153,Z 181.232,A -85,B 0,C 180,E1 -28771.095,E2 -28771.095} C_VEL
LIN {X 0,Y 58.523,Z 181.195,A -85,B 0,C 180,E1 -28783.878,E2 -28783.878} C_VEL
LIN {X 0,Y 58.815,Z 181.157,A -85,B 0,C 180,E1 -28793.14,E2 -28793.14} C_VEL
LIN {X 0,Y 59.391,Z 181.087,A -85,B 0,C 180,E1 -28800.003,E2 -28800.003} C_VEL
LIN {X 0,Y 58.821,Z 181.156,A -85,B 0,C 180,E1 -28806.865,E2 -28806.865} C_VEL
LIN {X 0,Y 58.655,Z 181.173,A -85,B 0,C 180,E1 -28813.868,E2 -28813.868} C_VEL
LIN {X 0,Y 58.163,Z 181.235,A -85,B 0,C 180,E1 -28826.947,E2 -28826.947} C_VEL
LIN {X 0,Y 58.161,Z 181.232,A -85,B 0,C 180,E1 -28827.923,E2 -28827.923} C_VEL
LIN {X 0,Y 59.245,Z 184.121,A -85,B 0,C 180,E1 -28829.386,E2 -28829.386} C_VEL
LIN {X 0,Y 60.654,Z 186.718,A -85,B 0,C 180,E1 -28830.831,E2 -28830.831} C_VEL
LIN {X 0,Y 65.006,Z 196.153,A -85,B 0,C 180,E1 -28835.057,E2 -28835.057} C_VEL
LIN {X 0,Y 68.001,Z 204.366,A -85,B 0,C 180,E1 -28837.901,E2 -28837.901} C_VEL
LIN {X 0,Y 72.026,Z 220.855,A -85,B 0,C 180,E1 -28842.177,E2 -28842.177} C_VEL
LIN {X 0,Y 72.638,Z 241.116,A -85,B 0,C 180,E1 -28845.69,E2 -28845.69} C_VEL
LIN {X 0,Y 68.753,Z 279.864,A -85,B 0,C 180,E1 -28851.474,E2 -28851.474} C_VEL
LIN {X 0,Y 66.817,Z 293.175,A -85,B 0,C 180,E1 -28854.658,E2 -28854.658} C_VEL
LIN {X 0,Y 64.479,Z 305.3,A -85,B 0,C 180,E1 -28858.823,E2 -28858.823} C_VEL
LIN {X 0,Y 62.176,Z 316.965,A -85,B 0,C 180,E1 -28864.337,E2 -28864.337} C_VEL
LIN {X 0,Y 60.264,Z 327.3,A -85,B 0,C 180,E1 -28870.794,E2 -28870.794} C_VEL
LIN {X 0,Y 59.26,Z 336.451,A -85,B 0,C 180,E1 -28878.024,E2 -28878.024} C_VEL
LIN {X 0,Y 59.003,Z 345.146,A -85,B 0,C 180,E1 -28886.588,E2 -28886.588} C_VEL
LIN {X 0,Y 59.735,Z 352.199,A -85,B 0,C 180,E1 -28895.065,E2 -28895.065} C_VEL
LIN {X 0,Y 59.831,Z 355.473,A -85,B 0,C 180,E1 -28900.151,E2 -28900.151} C_VEL
LIN {X 0,Y 60.914,Z 361.849,A -85,B 0,C 180,E1 -28912.625,E2 -28912.625} C_VEL
LIN {X 0,Y 64.391,Z 366.454,A -85,B 0,C 180,E1 -28923.077,E2 -28923.077} C_VEL
LIN {X 0,Y 71.366,Z 370.741,A -85,B 0,C 180,E1 -28933.582,E2 -28933.582} C_VEL
LIN {X 0,Y 80.573,Z 373.785,A -85,B 0,C 180,E1 -28941.726,E2 -28941.726} C_VEL
LIN {X 0,Y 92.634,Z 375.823,A -85,B 0,C 180,E1 -28948.534,E2 -28948.534} C_VEL
LIN {X 0,Y 93.938,Z 375.834,A -85,B 0,C 180,E1 -28950.087,E2 -28950.087} C_VEL
LIN {X 0,Y 83.832,Z 373.323,A -85,B 0,C 180,E1 -28955.216,E2 -28955.216} C_VEL
LIN {X 0,Y 73.181,Z 368.891,A -85,B 0,C 180,E1 -28963.253,E2 -28963.253} C_VEL
LIN {X 0,Y 64.714,Z 362.78,A -85,B 0,C 180,E1 -28973.763,E2 -28973.763} C_VEL
LIN {X 0,Y 59.686,Z 355.894,A -85,B 0,C 180,E1 -28985.064,E2 -28985.064} C_VEL
LIN {X 0,Y 57.467,Z 348.538,A -85,B 0,C 180,E1 -28995.969,E2 -28995.969} C_VEL
LIN {X 0,Y 57.108,Z 341.059,A -85,B 0,C 180,E1 -29005.511,E2 -29005.511} C_VEL
LIN {X 0,Y 57.611,Z 333.553,A -85,B 0,C 180,E1 -29013.491,E2 -29013.491} C_VEL
LIN {X 0,Y 59.001,Z 323.535,A -85,B 0,C 180,E1 -29022.066,E2 -29022.066} C_VEL
LIN {X 0,Y 61.079,Z 312.581,A -85,B 0,C 180,E1 -29029.283,E2 -29029.283} C_VEL
LIN {X 0,Y 61.236,Z 311.795,A -85,B 0,C 180,E1 -29029.719,E2 -29029.719} C_VEL
LIN {X 0,Y 61.604,Z 306.767,A -85,B 0,C 180,E1 -29032.411,E2 -29032.411} C_VEL
LIN {X 0,Y 60.536,Z 298.05,A -85,B 0,C 180,E1 -29036.629,E2 -29036.629} C_VEL
LIN {X 0,Y 59.455,Z 288.951,A -85,B 0,C 180,E1 -29040.488,E2 -29040.488} C_VEL
LIN {X 0,Y 59.825,Z 283.211,A -85,B 0,C 180,E1 -29042.409,E2 -29042.409} C_VEL
LIN {X 0,Y 61.882,Z 269.974,A -85,B 0,C 180,E1 -29045.547,E2 -29045.547} C_VEL
LIN {X 0,Y 67.1,Z 222.889,A -85,B 0,C 180,E1 -29052.758,E2 -29052.758} C_VEL
LIN {X 0,Y 61.39,Z 204.984,A -85,B 0,C 180,E1 -29058.646,E2 -29058.646} C_VEL
LIN {X 0,Y 56.332,Z 191.629,A -85,B 0,C 180,E1 -29064.366,E2 -29064.366} C_VEL
LIN {X 0,Y 52.384,Z 182.776,A -85,B 0,C 180,E1 -29069.516,E2 -29069.516} C_VEL
LIN {X 0,Y 52.282,Z 181.971,A -85,B 0,C 180,E1 -29069.997,E2 -29069.997} C_VEL
LIN {X 0,Y 51.69,Z 182.046,A -85,B 0,C 180,E1 -29077.811,E2 -29077.811} C_VEL
LIN {X 0,Y 51.391,Z 182.082,A -85,B 0,C 180,E1 -29086.816,E2 -29086.816} C_VEL
LIN {X 0,Y 51.025,Z 182.129,A -85,B 0,C 180,E1 -29094.404,E2 -29094.404} C_VEL
LIN {X 0,Y 51.049,Z 182.12,A -85,B 0,C 180,E1 -29104.312,E2 -29104.312} C_VEL
LIN {X 0,Y 51.056,Z 182.117,A -85,B 0,C 180,E1 -29113.488,E2 -29113.488} C_VEL
LIN {X 0,Y 51.056,Z 182.12,A -85,B 0,C 180,E1 -29116.512,E2 -29116.512} C_VEL
LIN {X 0,Y 51.071,Z 182.124,A -85,B 0,C 180,E1 -29126.606,E2 -29126.606} C_VEL
LIN {X 0,Y 51.025,Z 182.129,A -85,B 0,C 180,E1 -29135.597,E2 -29135.597} C_VEL
LIN {X 0,Y 51.464,Z 182.074,A -85,B 0,C 180,E1 -29144.153,E2 -29144.153} C_VEL
LIN {X 0,Y 51.69,Z 182.046,A -85,B 0,C 180,E1 -29152.189,E2 -29152.189} C_VEL
LIN {X 0,Y 52.276,Z 181.974,A -85,B 0,C 180,E1 -29160.003,E2 -29160.003} C_VEL
LIN {X 0,Y 51.697,Z 182.046,A -85,B 0,C 180,E1 -29167.816,E2 -29167.816} C_VEL
LIN {X 0,Y 51.371,Z 182.086,A -85,B 0,C 180,E1 -29176.742,E2 -29176.742} C_VEL
LIN {X 0,Y 51.137,Z 182.111,A -85,B 0,C 180,E1 -29182.876,E2 -29182.876} C_VEL
LIN {X 0,Y 52.04,Z 184.794,A -85,B 0,C 180,E1 -29184.434,E2 -29184.434} C_VEL
LIN {X 0,Y 53.544,Z 187.372,A -85,B 0,C 180,E1 -29186.298,E2 -29186.298} C_VEL
LIN {X 0,Y 56.559,Z 193.297,A -85,B 0,C 180,E1 -29189.808,E2 -29189.808} C_VEL
LIN {X 0,Y 60.53,Z 202.811,A -85,B 0,C 180,E1 -29194.168,E2 -29194.168} C_VEL
LIN {X 0,Y 62.217,Z 208.281,A -85,B 0,C 180,E1 -29196.125,E2 -29196.125} C_VEL
LIN {X 0,Y 65.505,Z 223.09,A -85,B 0,C 180,E1 -29200.369,E2 -29200.369} C_VEL
LIN {X 0,Y 65.856,Z 241.717,A -85,B 0,C 180,E1 -29203.92,E2 -29203.92} C_VEL
LIN {X 0,Y 61.892,Z 279.294,A -85,B 0,C 180,E1 -29210.041,E2 -29210.041} C_VEL
LIN {X 0,Y 59.863,Z 292.617,A -85,B 0,C 180,E1 -29213.537,E2 -29213.537} C_VEL
LIN {X 0,Y 57.265,Z 305.646,A -85,B 0,C 180,E1 -29218.564,E2 -29218.564} C_VEL
LIN {X 0,Y 54.981,Z 316.93,A -85,B 0,C 180,E1 -29224.643,E2 -29224.643} C_VEL
LIN {X 0,Y 52.986,Z 328.069,A -85,B 0,C 180,E1 -29232.74,E2 -29232.74} C_VEL
LIN {X 0,Y 52.262,Z 338.105,A -85,B 0,C 180,E1 -29242.275,E2 -29242.275} C_VEL
LIN {X 0,Y 52.859,Z 347.789,A -85,B 0,C 180,E1 -29253.815,E2 -29253.815} C_VEL
LIN {X 0,Y 53.392,Z 351.65,A -85,B 0,C 180,E1 -29259.473,E2 -29259.473} C_VEL
LIN {X 0,Y 53.738,Z 356.59,A -85,B 0,C 180,E1 -29269.087,E2 -29269.087} C_VEL
LIN {X 0,Y 57.364,Z 362.989,A -85,B 0,C 180,E1 -29283.461,E2 -29283.461} C_VEL
LIN {X 0,Y 64.388,Z 367.974,A -85,B 0,C 180,E1 -29295.196,E2 -29295.196} C_VEL
LIN {X 0,Y 71.276,Z 370.824,A -85,B 0,C 180,E1 -29302.078,E2 -29302.078} C_VEL
LIN {X 0,Y 81.95,Z 373.646,A -85,B 0,C 180,E1 -29309.051,E2 -29309.051} C_VEL
LIN {X 0,Y 80.587,Z 373.106,A -85,B 0,C 180,E1 -29310.708,E2 -29310.708} C_VEL
LIN {X 0,Y 69.225,Z 368.454,A -85,B 0,C 180,E1 -29318.353,E2 -29318.353} C_VEL
LIN {X 0,Y 61.285,Z 363.431,A -85,B 0,C 180,E1 -29326.738,E2 -29326.738} C_VEL
LIN {X 0,Y 54.814,Z 356.541,A -85,B 0,C 180,E1 -29338.305,E2 -29338.305} C_VEL
LIN {X 0,Y 51.398,Z 349.245,A -85,B 0,C 180,E1 -29350.168,E2 -29350.168} C_VEL
LIN {X 0,Y 50.388,Z 342.349,A -85,B 0,C 180,E1 -29360.404,E2 -29360.404} C_VEL
LIN {X 0,Y 50.631,Z 333.391,A -85,B 0,C 180,E1 -29371.365,E2 -29371.365} C_VEL
LIN {X 0,Y 51.878,Z 323.088,A -85,B 0,C 180,E1 -29381.327,E2 -29381.327} C_VEL
LIN {X 0,Y 53.926,Z 312.369,A -85,B 0,C 180,E1 -29389.332,E2 -29389.332} C_VEL
LIN {X 0,Y 56.561,Z 299.895,A -85,B 0,C 180,E1 -29396.193,E2 -29396.193} C_VEL
LIN {X 0,Y 59.091,Z 287.398,A -85,B 0,C 180,E1 -29401.134,E2 -29401.134} C_VEL
LIN {X 0,Y 59.825,Z 283.211,A -85,B 0,C 180,E1 -29402.409,E2 -29402.409} C_VEL
LIN {X 0,Y 60.134,Z 277.573,A -85,B 0,C 180,E1 -29404.074,E2 -29404.074} C_VEL
LIN {X 0,Y 58.682,Z 268.172,A -85,B 0,C 180,E1 -29406.793,E2 -29406.793} C_VEL
LIN {X 0,Y 57.002,Z 258.662,A -85,B 0,C 180,E1 -29409.292,E2 -29409.292} C_VEL
LIN {X 0,Y 57.037,Z 252.841,A -85,B 0,C 180,E1 -29410.48,E2 -29410.48} C_VEL
LIN {X 0,Y 60.454,Z 224.249,A -85,B 0,C 180,E1 -29415.12,E2 -29415.12} C_VEL
LIN {X 0,Y 55.235,Z 207.296,A -85,B 0,C 180,E1 -29421.384,E2 -29421.384} C_VEL
LIN {X 0,Y 50.78,Z 195.04,A -85,B 0,C 180,E1 -29427.533,E2 -29427.533} C_VEL
LIN {X 0,Y 47.353,Z 187.432,A -85,B 0,C 180,E1 -29432.838,E2 -29432.838} C_VEL
LIN {X 0,Y 45.307,Z 185.001,A -85,B 0,C 180,E1 -29435.839,E2 -29435.839} C_VEL
LIN {X 0,Y 44.651,Z 182.923,A -85,B 0,C 180,E1 -29437.344,E2 -29437.344} C_VEL
LIN {X 0,Y 44.154,Z 182.977,A -85,B 0,C 180,E1 -29448.559,E2 -29448.559} C_VEL
LIN {X 0,Y 43.853,Z 183.014,A -85,B 0,C 180,E1 -29458.733,E2 -29458.733} C_VEL
LIN {X 0,Y 43.866,Z 183.021,A -85,B 0,C 180,E1 -29469.852,E2 -29469.852} C_VEL
LIN {X 0,Y 43.887,Z 183.009,A -85,B 0,C 180,E1 -29483.19,E2 -29483.19} C_VEL
LIN {X 0,Y 43.853,Z 183.013,A -85,B 0,C 180,E1 -29491.267,E2 -29491.267} C_VEL
LIN {X 0,Y 44.229,Z 182.974,A -85,B 0,C 180,E1 -29502.428,E2 -29502.428} C_VEL
LIN {X 0,Y 44.541,Z 182.936,A -85,B 0,C 180,E1 -29510.925,E2 -29510.925} C_VEL
LIN {X 0,Y 45.151,Z 182.861,A -85,B 0,C 180,E1 -29520.003,E2 -29520.003} C_VEL
LIN {X 0,Y 44.395,Z 182.947,A -85,B 0,C 180,E1 -29533.74,E2 -29533.74} C_VEL
LIN {X 0,Y 44.368,Z 183.087,A -85,B 0,C 180,E1 -29536.028,E2 -29536.028} C_VEL
LIN {X 0,Y 45.264,Z 185.864,A -85,B 0,C 180,E1 -29538.095,E2 -29538.095} C_VEL
LIN {X 0,Y 46.799,Z 188.37,A -85,B 0,C 180,E1 -29540.611,E2 -29540.611} C_VEL
LIN {X 0,Y 50.77,Z 196.17,A -85,B 0,C 180,E1 -29546.463,E2 -29546.463} C_VEL
LIN {X 0,Y 54.667,Z 205.841,A -85,B 0,C 180,E1 -29551.582,E2 -29551.582} C_VEL
LIN {X 0,Y 56.501,Z 212.364,A -85,B 0,C 180,E1 -29554.107,E2 -29554.107} C_VEL
LIN {X 0,Y 59.017,Z 224.709,A -85,B 0,C 180,E1 -29558.02,E2 -29558.02} C_VEL
LIN {X 0,Y 59.173,Z 242.491,A -85,B 0,C 180,E1 -29561.792,E2 -29561.792} C_VEL
LIN {X 0,Y 54.948,Z 279.51,A -85,B 0,C 180,E1 -29568.437,E2 -29568.437} C_VEL
LIN {X 0,Y 52.786,Z 292.667,A -85,B 0,C 180,E1 -29572.357,E2 -29572.357} C_VEL
LIN {X 0,Y 50.305,Z 304.662,A -85,B 0,C 180,E1 -29577.629,E2 -29577.629} C_VEL
LIN {X 0,Y 47.845,Z 316.584,A -85,B 0,C 180,E1 -29585.023,E2 -29585.023} C_VEL
LIN {X 0,Y 45.944,Z 327.706,A -85,B 0,C 180,E1 -29594.476,E2 -29594.476} C_VEL
LIN {X 0,Y 45.512,Z 337.771,A -85,B 0,C 180,E1 -29605.575,E2 -29605.575} C_VEL
LIN {X 0,Y 46.42,Z 345.913,A -85,B 0,C 180,E1 -29616.523,E2 -29616.523} C_VEL
LIN {X 0,Y 46.961,Z 348.655,A -85,B 0,C 180,E1 -29620.785,E2 -29620.785} C_VEL
LIN {X 0,Y 47.59,Z 353.869,A -85,B 0,C 180,E1 -29631.67,E2 -29631.67} C_VEL
LIN {X 0,Y 51.92,Z 360.637,A -85,B 0,C 180,E1 -29647.53,E2 -29647.53} C_VEL
LIN {X 0,Y 59.786,Z 365.935,A -85,B 0,C 180,E1 -29659.83,E2 -29659.83} C_VEL
LIN {X 0,Y 67.256,Z 369.096,A -85,B 0,C 180,E1 -29666.721,E2 -29666.721} C_VEL
LIN {X 0,Y 70.17,Z 369.945,A -85,B 0,C 180,E1 -29669.946,E2 -29669.946} C_VEL
LIN {X 0,Y 58.9,Z 363.96,A -85,B 0,C 180,E1 -29679.022,E2 -29679.022} C_VEL
LIN {X 0,Y 50.973,Z 357.327,A -85,B 0,C 180,E1 -29690.073,E2 -29690.073} C_VEL
LIN {X 0,Y 45.661,Z 348.984,A -85,B 0,C 180,E1 -29704.41,E2 -29704.41} C_VEL
LIN {X 0,Y 43.735,Z 340.202,A -85,B 0,C 180,E1 -29718.743,E2 -29718.743} C_VEL
LIN {X 0,Y 43.78,Z 331.147,A -85,B 0,C 180,E1 -29731.124,E2 -29731.124} C_VEL
LIN {X 0,Y 44.978,Z 321.314,A -85,B 0,C 180,E1 -29741.608,E2 -29741.608} C_VEL
LIN {X 0,Y 47.333,Z 309.367,A -85,B 0,C 180,E1 -29751.246,E2 -29751.246} C_VEL
LIN {X 0,Y 50.029,Z 297.063,A -85,B 0,C 180,E1 -29758.387,E2 -29758.387} C_VEL
LIN {X 0,Y 52.566,Z 284.749,A -85,B 0,C 180,E1 -29763.388,E2 -29763.388} C_VEL
LIN {X 0,Y 54.882,Z 271.034,A -85,B 0,C 180,E1 -29767.172,E2 -29767.172} C_VEL
LIN {X 0,Y 57.037,Z 252.841,A -85,B 0,C 180,E1 -29770.48,E2 -29770.48} C_VEL
LIN {X 0,Y 56.852,Z 248.953,A -85,B 0,C 180,E1 -29771.366,E2 -29771.366} C_VEL
LIN {X 0,Y 52.999,Z 236.671,A -85,B 0,C 180,E1 -29775.702,E2 -29775.702} C_VEL
LIN {X 0,Y 52.947,Z 232.788,A -85,B 0,C 180,E1 -29776.636,E2 -29776.636} C_VEL
LIN {X 0,Y 53.766,Z 224.938,A -85,B 0,C 180,E1 -29778.058,E2 -29778.058} C_VEL
LIN {X 0,Y 48.835,Z 208.29,A -85,B 0,C 180,E1 -29785.468,E2 -29785.468} C_VEL
LIN {X 0,Y 45.242,Z 198.013,A -85,B 0,C 180,E1 -29791.68,E2 -29791.68} C_VEL
LIN {X 0,Y 42.98,Z 192.628,A -85,B 0,C 180,E1 -29795.951,E2 -29795.951} C_VEL
LIN {X 0,Y 40.76,Z 189.424,A -85,B 0,C 180,E1 -29800.12,E2 -29800.12} C_VEL
LIN {X 0,Y 39.927,Z 188.486,A -85,B 0,C 180,E1 -29801.785,E2 -29801.785} C_VEL
LIN {X 0,Y 38.021,Z 186.382,A -85,B 0,C 180,E1 -29806.098,E2 -29806.098} C_VEL
LIN {X 0,Y 36.968,Z 183.871,A -85,B 0,C 180,E1 -29809.912,E2 -29809.912} C_VEL
LIN {X 0,Y 36.753,Z 183.898,A -85,B 0,C 180,E1 -29825.001,E2 -29825.001} C_VEL
LIN {X 0,Y 36.777,Z 183.904,A -85,B 0,C 180,E1 -29830.153,E2 -29830.153} C_VEL
LIN {X 0,Y 36.777,Z 183.9,A -85,B 0,C 180,E1 -29839.847,E2 -29839.847} C_VEL
LIN {X 0,Y 36.754,Z 183.901,A -85,B 0,C 180,E1 -29845,E2 -29845} C_VEL
LIN {X 0,Y 37.056,Z 183.863,A -85,B 0,C 180,E1 -29861.482,E2 -29861.482} C_VEL
LIN {X 0,Y 37.334,Z 183.827,A -85,B 0,C 180,E1 -29869.154,E2 -29869.154} C_VEL
LIN {X 0,Y 38.009,Z 183.751,A -85,B 0,C 180,E1 -29880.004,E2 -29880.004} C_VEL
LIN {X 0,Y 37.621,Z 183.79,A -85,B 0,C 180,E1 -29885.364,E2 -29885.364} C_VEL
LIN {X 0,Y 38.462,Z 186.589,A -85,B 0,C 180,E1 -29888.542,E2 -29888.542} C_VEL
LIN {X 0,Y 40.154,Z 188.867,A -85,B 0,C 180,E1 -29892.381,E2 -29892.381} C_VEL
LIN {X 0,Y 44.838,Z 198.228,A -85,B 0,C 180,E1 -29901.67,E2 -29901.67} C_VEL
LIN {X 0,Y 48.737,Z 208.304,A -85,B 0,C 180,E1 -29908.17,E2 -29908.17} C_VEL
LIN {X 0,Y 50.445,Z 214.73,A -85,B 0,C 180,E1 -29911.098,E2 -29911.098} C_VEL
LIN {X 0,Y 52.575,Z 225.329,A -85,B 0,C 180,E1 -29915.028,E2 -29915.028} C_VEL
LIN {X 0,Y 52.587,Z 242.504,A -85,B 0,C 180,E1 -29919.103,E2 -29919.103} C_VEL
LIN {X 0,Y 48.118,Z 279.049,A -85,B 0,C 180,E1 -29926.437,E2 -29926.437} C_VEL
LIN {X 0,Y 45.952,Z 291.521,A -85,B 0,C 180,E1 -29930.591,E2 -29930.591} C_VEL
LIN {X 0,Y 43.269,Z 303.919,A -85,B 0,C 180,E1 -29936.715,E2 -29936.715} C_VEL
LIN {X 0,Y 40.919,Z 314.988,A -85,B 0,C 180,E1 -29944.576,E2 -29944.576} C_VEL
LIN {X 0,Y 39.046,Z 326.33,A -85,B 0,C 180,E1 -29955.675,E2 -29955.675} C_VEL
LIN {X 0,Y 38.835,Z 335.644,A -85,B 0,C 180,E1 -29967.411,E2 -29967.411} C_VEL
LIN {X 0,Y 40.161,Z 343.955,A -85,B 0,C 180,E1 -29980.082,E2 -29980.082} C_VEL
LIN {X 0,Y 40.813,Z 346.686,A -85,B 0,C 180,E1 -29984.973,E2 -29984.973} C_VEL
LIN {X 0,Y 42.551,Z 352.925,A -85,B 0,C 180,E1 -29999.707,E2 -29999.707} C_VEL
LIN {X 0,Y 46.839,Z 358.127,A -85,B 0,C 180,E1 -30012.469,E2 -30012.469} C_VEL
LIN {X 0,Y 55.662,Z 363.782,A -85,B 0,C 180,E1 -30025.16,E2 -30025.16} C_VEL
LIN {X 0,Y 58.254,Z 365.002,A -85,B 0,C 180,E1 -30027.623,E2 -30027.623} C_VEL
LIN {X 0,Y 58.935,Z 365.186,A -85,B 0,C 180,E1 -30029.79,E2 -30029.79} C_VEL
LIN {X 0,Y 48.24,Z 357.865,A -85,B 0,C 180,E1 -30040.862,E2 -30040.862} C_VEL
LIN {X 0,Y 41.122,Z 349.744,A -85,B 0,C 180,E1 -30055.089,E2 -30055.089} C_VEL
LIN {X 0,Y 37.707,Z 341.198,A -85,B 0,C 180,E1 -30070.738,E2 -30070.738} C_VEL
LIN {X 0,Y 36.904,Z 332.302,A -85,B 0,C 180,E1 -30085.367,E2 -30085.367} C_VEL
LIN {X 0,Y 37.695,Z 322.412,A -85,B 0,C 180,E1 -30098.542,E2 -30098.542} C_VEL
LIN {X 0,Y 39.899,Z 310.492,A -85,B 0,C 180,E1 -30110.405,E2 -30110.405} C_VEL
LIN {X 0,Y 42.635,Z 298.309,A -85,B 0,C 180,E1 -30118.902,E2 -30118.902} C_VEL
LIN {X 0,Y 45.393,Z 285.75,A -85,B 0,C 180,E1 -30124.858,E2 -30124.858} C_VEL
LIN {X 0,Y 47.916,Z 271.858,A -85,B 0,C 180,E1 -30129.227,E2 -30129.227} C_VEL
LIN {X 0,Y 52.947,Z 232.788,A -85,B 0,C 180,E1 -30136.636,E2 -30136.636} C_VEL
LIN {X 0,Y 52.782,Z 229.697,A -85,B 0,C 180,E1 -30137.455,E2 -30137.455} C_VEL
LIN {X 0,Y 51.084,Z 225.805,A -85,B 0,C 180,E1 -30139.353,E2 -30139.353} C_VEL
LIN {X 0,Y 45.089,Z 217.176,A -85,B 0,C 180,E1 -30145.951,E2 -30145.951} C_VEL
LIN {X 0,Y 44.387,Z 215.39,A -85,B 0,C 180,E1 -30147.069,E2 -30147.069} C_VEL
LIN {X 0,Y 40.656,Z 202.987,A -85,B 0,C 180,E1 -30155.051,E2 -30155.051} C_VEL
LIN {X 0,Y 38.63,Z 197.594,A -85,B 0,C 180,E1 -30159.981,E2 -30159.981} C_VEL
LIN {X 0,Y 36.433,Z 194.321,A -85,B 0,C 180,E1 -30165.324,E2 -30165.324} C_VEL
LIN {X 0,Y 34.353,Z 191.415,A -85,B 0,C 180,E1 -30171.543,E2 -30171.543} C_VEL
LIN {X 0,Y 33.894,Z 190.399,A -85,B 0,C 180,E1 -30173.363,E2 -30173.363} C_VEL
LIN {X 0,Y 31.257,Z 188.492,A -85,B 0,C 180,E1 -30183.879,E2 -30183.879} C_VEL
LIN {X 0,Y 29.742,Z 185.024,A -85,B 0,C 180,E1 -30201.669,E2 -30201.669} C_VEL
LIN {X 0,Y 29.616,Z 185.128,A -85,B 0,C 180,E1 -30207.734,E2 -30207.734} C_VEL
LIN {X 0,Y 30.464,Z 186.434,A -85,B 0,C 180,E1 -30223.084,E2 -30223.084} C_VEL
LIN {X 0,Y 33.724,Z 189.539,A -85,B 0,C 180,E1 -30239.258,E2 -30239.258} C_VEL
LIN {X 0,Y 34.175,Z 189.995,A -85,B 0,C 180,E1 -30240.814,E2 -30240.814} C_VEL
LIN {X 0,Y 35.925,Z 193.612,A -85,B 0,C 180,E1 -30247.023,E2 -30247.023} C_VEL
LIN {X 0,Y 38.899,Z 199.979,A -85,B 0,C 180,E1 -30255.057,E2 -30255.057} C_VEL
LIN {X 0,Y 41.737,Z 207.069,A -85,B 0,C 180,E1 -30261.248,E2 -30261.248} C_VEL
LIN {X 0,Y 44.126,Z 214.893,A -85,B 0,C 180,E1 -30266.216,E2 -30266.216} C_VEL
LIN {X 0,Y 46.281,Z 226.793,A -85,B 0,C 180,E1 -30271.505,E2 -30271.505} C_VEL
LIN {X 0,Y 46.066,Z 242.808,A -85,B 0,C 180,E1 -30275.822,E2 -30275.822} C_VEL
LIN {X 0,Y 41.375,Z 278.37,A -85,B 0,C 180,E1 -30283.723,E2 -30283.723} C_VEL
LIN {X 0,Y 38.961,Z 291.323,A -85,B 0,C 180,E1 -30288.631,E2 -30288.631} C_VEL
LIN {X 0,Y 36.502,Z 302.124,A -85,B 0,C 180,E1 -30294.722,E2 -30294.722} C_VEL
LIN {X 0,Y 34.008,Z 313.379,A -85,B 0,C 180,E1 -30303.956,E2 -30303.956} C_VEL
LIN {X 0,Y 32.177,Z 325.964,A -85,B 0,C 180,E1 -30318.987,E2 -30318.987} C_VEL
LIN {X 0,Y 32.495,Z 335.092,A -85,B 0,C 180,E1 -30333.104,E2 -30333.104} C_VEL
LIN {X 0,Y 34.65,Z 343.312,A -85,B 0,C 180,E1 -30347.717,E2 -30347.717} C_VEL
LIN {X 0,Y 35.544,Z 346.848,A -85,B 0,C 180,E1 -30356.42,E2 -30356.42} C_VEL
LIN {X 0,Y 40.258,Z 353.715,A -85,B 0,C 180,E1 -30374.295,E2 -30374.295} C_VEL
LIN {X 0,Y 47.693,Z 359.133,A -85,B 0,C 180,E1 -30386.679,E2 -30386.679} C_VEL
LIN {X 0,Y 49.017,Z 359.833,A -85,B 0,C 180,E1 -30388.769,E2 -30388.769} C_VEL
LIN {X 0,Y 40.236,Z 352.806,A -85,B 0,C 180,E1 -30399.549,E2 -30399.549} C_VEL
LIN {X 0,Y 34.062,Z 344.987,A -85,B 0,C 180,E1 -30414.074,E2 -30414.074} C_VEL
LIN {X 0,Y 31.075,Z 337.235,A -85,B 0,C 180,E1 -30429.761,E2 -30429.761} C_VEL
LIN {X 0,Y 30.246,Z 329.085,A -85,B 0,C 180,E1 -30444.76,E2 -30444.76} C_VEL
LIN {X 0,Y 31.069,Z 318.595,A -85,B 0,C 180,E1 -30460.561,E2 -30460.561} C_VEL
LIN {X 0,Y 33.5,Z 306.668,A -85,B 0,C 180,E1 -30473.602,E2 -30473.602} C_VEL
LIN {X 0,Y 36.515,Z 294.156,A -85,B 0,C 180,E1 -30482.885,E2 -30482.885} C_VEL
LIN {X 0,Y 39.478,Z 280.957,A -85,B 0,C 180,E1 -30489.215,E2 -30489.215} C_VEL
LIN {X 0,Y 41.903,Z 267.214,A -85,B 0,C 180,E1 -30493.32,E2 -30493.32} C_VEL
LIN {X 0,Y 47.431,Z 226.463,A -85,B 0,C 180,E1 -30501.476,E2 -30501.476} C_VEL
LIN {X 0,Y 44.387,Z 215.39,A -85,B 0,C 180,E1 -30507.069,E2 -30507.069} C_VEL
LIN {X 0,Y 42.907,Z 212.213,A -85,B 0,C 180,E1 -30509.414,E2 -30509.414} C_VEL
LIN {X 0,Y 39.427,Z 208.053,A -85,B 0,C 180,E1 -30514.721,E2 -30514.721} C_VEL
LIN {X 0,Y 34.126,Z 201.918,A -85,B 0,C 180,E1 -30526.176,E2 -30526.176} C_VEL
LIN {X 0,Y 32.959,Z 199.952,A -85,B 0,C 180,E1 -30529.98,E2 -30529.98} C_VEL
LIN {X 0,Y 31.071,Z 196.767,A -85,B 0,C 180,E1 -30537.524,E2 -30537.524} C_VEL
LIN {X 0,Y 28.805,Z 194.213,A -85,B 0,C 180,E1 -30551.265,E2 -30551.265} C_VEL
LIN {X 0,Y 28.32,Z 191.919,A -85,B 0,C 180,E1 -30564.54,E2 -30564.54} C_VEL
LIN {X 0,Y 28.662,Z 193.077,A -85,B 0,C 180,E1 -30579.396,E2 -30579.396} C_VEL
LIN {X 0,Y 31.188,Z 196.149,A -85,B 0,C 180,E1 -30595.967,E2 -30595.967} C_VEL
LIN {X 0,Y 33.026,Z 200.59,A -85,B 0,C 180,E1 -30604.298,E2 -30604.298} C_VEL
LIN {X 0,Y 35.565,Z 207.268,A -85,B 0,C 180,E1 -30612.985,E2 -30612.985} C_VEL
LIN {X 0,Y 38.021,Z 215.409,A -85,B 0,C 180,E1 -30619.974,E2 -30619.974} C_VEL
LIN {X 0,Y 39.758,Z 225.216,A -85,B 0,C 180,E1 -30625.474,E2 -30625.474} C_VEL
LIN {X 0,Y 40.178,Z 229.002,A -85,B 0,C 180,E1 -30627.157,E2 -30627.157} C_VEL
LIN {X 0,Y 39.785,Z 242.788,A -85,B 0,C 180,E1 -30631.404,E2 -30631.404} C_VEL
LIN {X 0,Y 34.728,Z 277.744,A -85,B 0,C 180,E1 -30640.081,E2 -30640.081} C_VEL
LIN {X 0,Y 32.399,Z 289.532,A -85,B 0,C 180,E1 -30645.178,E2 -30645.178} C_VEL
LIN {X 0,Y 29.42,Z 301.743,A -85,B 0,C 180,E1 -30653.336,E2 -30653.336} C_VEL
LIN {X 0,Y 26.905,Z 312.89,A -85,B 0,C 180,E1 -30664.889,E2 -30664.889} C_VEL
LIN {X 0,Y 25.447,Z 325.421,A -85,B 0,C 180,E1 -30684.061,E2 -30684.061} C_VEL
LIN {X 0,Y 26.628,Z 334.525,A -85,B 0,C 180,E1 -30701.423,E2 -30701.423} C_VEL
LIN {X 0,Y 29.145,Z 341.139,A -85,B 0,C 180,E1 -30714.966,E2 -30714.966} C_VEL
LIN {X 0,Y 33.835,Z 348.804,A -85,B 0,C 180,E1 -30736.642,E2 -30736.642} C_VEL
LIN {X 0,Y 39.244,Z 353.282,A -85,B 0,C 180,E1 -30747.499,E2 -30747.499} C_VEL
LIN {X 0,Y 30.315,Z 344.485,A -85,B 0,C 180,E1 -30762.516,E2 -30762.516} C_VEL
LIN {X 0,Y 25.048,Z 334.578,A -85,B 0,C 180,E1 -30784.016,E2 -30784.016} C_VEL
LIN {X 0,Y 23.671,Z 326.271,A -85,B 0,C 180,E1 -30802.391,E2 -30802.391} C_VEL
LIN {X 0,Y 24.272,Z 316.358,A -85,B 0,C 180,E1 -30820.646,E2 -30820.646} C_VEL
LIN {X 0,Y 26.883,Z 304.222,A -85,B 0,C 180,E1 -30836.561,E2 -30836.561} C_VEL
LIN {X 0,Y 30.401,Z 290.56,A -85,B 0,C 180,E1 -30847.612,E2 -30847.612} C_VEL
LIN {X 0,Y 33.54,Z 276.87,A -85,B 0,C 180,E1 -30854.257,E2 -30854.257} C_VEL
LIN {X 0,Y 36.051,Z 261.954,A -85,B 0,C 180,E1 -30858.523,E2 -30858.523} C_VEL
LIN {X 0,Y 41.113,Z 227.484,A -85,B 0,C 180,E1 -30866.073,E2 -30866.073} C_VEL
LIN {X 0,Y 37.217,Z 212.008,A -85,B 0,C 180,E1 -30876.071,E2 -30876.071} C_VEL
LIN {X 0,Y 35.138,Z 204.389,A -85,B 0,C 180,E1 -30882.853,E2 -30882.853} C_VEL
LIN {X 0,Y 34.303,Z 202.174,A -85,B 0,C 180,E1 -30885.658,E2 -30885.658} C_VEL
LIN {X 0,Y 34.126,Z 201.918,A -85,B 0,C 180,E1 -30886.176,E2 -30886.176} C_VEL
LIN {X 0,Y 32.466,Z 200.005,A -85,B 0,C 180,E1 -30891.256,E2 -30891.256} C_VEL
LIN {X 0,Y 30.072,Z 199.049,A -85,B 0,C 180,E1 -30899.722,E2 -30899.722} C_VEL
LIN {X 0,Y 26.868,Z 199.329,A -85,B 0,C 180,E1 -30924.458,E2 -30924.458} C_VEL
LIN {X 0,Y 26.952,Z 199.532,A -85,B 0,C 180,E1 -30933.908,E2 -30933.908} C_VEL
LIN {X 0,Y 28.58,Z 202.561,A -85,B 0,C 180,E1 -30951.164,E2 -30951.164} C_VEL
LIN {X 0,Y 29.929,Z 206.741,A -85,B 0,C 180,E1 -30959.637,E2 -30959.637} C_VEL
LIN {X 0,Y 31.554,Z 212.589,A -85,B 0,C 180,E1 -30967.811,E2 -30967.811} C_VEL
LIN {X 0,Y 33.217,Z 220.052,A -85,B 0,C 180,E1 -30975.015,E2 -30975.015} C_VEL
LIN {X 0,Y 34.33,Z 230.104,A -85,B 0,C 180,E1 -30981.199,E2 -30981.199} C_VEL
LIN {X 0,Y 33.652,Z 242.999,A -85,B 0,C 180,E1 -30985.724,E2 -30985.724} C_VEL
LIN {X 0,Y 28.038,Z 278.088,A -85,B 0,C 180,E1 -30995.457,E2 -30995.457} C_VEL
LIN {X 0,Y 25.322,Z 290.21,A -85,B 0,C 180,E1 -31001.771,E2 -31001.771} C_VEL
LIN {X 0,Y 21.946,Z 303.009,A -85,B 0,C 180,E1 -31013.106,E2 -31013.106} C_VEL
LIN {X 0,Y 19.281,Z 315.072,A -85,B 0,C 180,E1 -31031.41,E2 -31031.41} C_VEL
LIN {X 0,Y 19.237,Z 325.998,A -85,B 0,C 180,E1 -31055.248,E2 -31055.248} C_VEL
LIN {X 0,Y 22.509,Z 335.566,A -85,B 0,C 180,E1 -31077.934,E2 -31077.934} C_VEL
LIN {X 0,Y 24.346,Z 338.757,A -85,B 0,C 180,E1 -31085.272,E2 -31085.272} C_VEL
LIN {X 0,Y 27.66,Z 343.403,A -85,B 0,C 180,E1 -31099.671,E2 -31099.671} C_VEL
LIN {X 0,Y 29.604,Z 345.342,A -85,B 0,C 180,E1 -31105.923,E2 -31105.923} C_VEL
LIN {X 0,Y 22.07,Z 336.617,A -85,B 0,C 180,E1 -31122.831,E2 -31122.831} C_VEL
LIN {X 0,Y 18.082,Z 327.801,A -85,B 0,C 180,E1 -31145.568,E2 -31145.568} C_VEL
LIN {X 0,Y 17.135,Z 317.606,A -85,B 0,C 180,E1 -31172.216,E2 -31172.216} C_VEL
LIN {X 0,Y 19.245,Z 305.92,A -85,B 0,C 180,E1 -31195.237,E2 -31195.237} C_VEL
LIN {X 0,Y 22.543,Z 294.003,A -85,B 0,C 180,E1 -31209.255,E2 -31209.255} C_VEL
LIN {X 0,Y 26.319,Z 279.809,A -85,B 0,C 180,E1 -31218.313,E2 -31218.313} C_VEL
LIN {X 0,Y 29.087,Z 265.99,A -85,B 0,C 180,E1 -31223.183,E2 -31223.183} C_VEL
LIN {X 0,Y 35.14,Z 228.915,A -85,B 0,C 180,E1 -31231.88,E2 -31231.88} C_VEL
LIN {X 0,Y 32.336,Z 215.163,A -85,B 0,C 180,E1 -31242.83,E2 -31242.83} C_VEL
LIN {X 0,Y 30.781,Z 207.783,A -85,B 0,C 180,E1 -31250.727,E2 -31250.727} C_VEL
LIN {X 0,Y 29.578,Z 205.306,A -85,B 0,C 180,E1 -31256.075,E2 -31256.075} C_VEL
LIN {X 0,Y 28.273,Z 202.944,A -85,B 0,C 180,E1 -31263.505,E2 -31263.505} C_VEL
LIN {X 0,Y 26.868,Z 199.329,A -85,B 0,C 180,E1 -31284.458,E2 -31284.458} C_VEL
LIN {X 0,Y 26.753,Z 199.968,A -85,B 0,C 180,E1 -31291.07,E2 -31291.07} C_VEL
LIN {X 0,Y 26.718,Z 202.156,A -85,B 0,C 180,E1 -31298.016,E2 -31298.016} C_VEL
LIN {X 0,Y 26.728,Z 204.628,A -85,B 0,C 180,E1 -31302.792,E2 -31302.792} C_VEL
LIN {X 0,Y 27.235,Z 214.519,A -85,B 0,C 180,E1 -31316.49,E2 -31316.49} C_VEL
LIN {X 0,Y 28.371,Z 221.699,A -85,B 0,C 180,E1 -31325.518,E2 -31325.518} C_VEL
LIN {X 0,Y 28.973,Z 231.67,A -85,B 0,C 180,E1 -31333.152,E2 -31333.152} C_VEL
LIN {X 0,Y 28.048,Z 242.907,A -85,B 0,C 180,E1 -31337.619,E2 -31337.619} C_VEL
LIN {X 0,Y 21.822,Z 277.644,A -85,B 0,C 180,E1 -31347.681,E2 -31347.681} C_VEL
LIN {X 0,Y 18.73,Z 289.713,A -85,B 0,C 180,E1 -31354.847,E2 -31354.847} C_VEL
LIN {X 0,Y 14.93,Z 302.456,A -85,B 0,C 180,E1 -31369.679,E2 -31369.679} C_VEL
LIN {X 0,Y 12.362,Z 314.348,A -85,B 0,C 180,E1 -31397.702,E2 -31397.702} C_VEL
LIN {X 0,Y 13.961,Z 325.181,A -85,B 0,C 180,E1 -31432.193,E2 -31432.193} C_VEL
LIN {X 0,Y 19.537,Z 334.755,A -85,B 0,C 180,E1 -31456.019,E2 -31456.019} C_VEL
LIN {X 0,Y 20.378,Z 335.964,A -85,B 0,C 180,E1 -31462.904,E2 -31462.904} C_VEL
LIN {X 0,Y 14.51,Z 328.344,A -85,B 0,C 180,E1 -31480.525,E2 -31480.525} C_VEL
LIN {X 0,Y 10.993,Z 319.741,A -85,B 0,C 180,E1 -31509.183,E2 -31509.183} C_VEL
LIN {X 0,Y 11.446,Z 308.044,A -85,B 0,C 180,E1 -31550.064,E2 -31550.064} C_VEL
LIN {X 0,Y 15.099,Z 295.763,A -85,B 0,C 180,E1 -31573.713,E2 -31573.713} C_VEL
LIN {X 0,Y 19.175,Z 282.686,A -85,B 0,C 180,E1 -31585.103,E2 -31585.103} C_VEL
LIN {X 0,Y 22.695,Z 268.383,A -85,B 0,C 180,E1 -31590.992,E2 -31590.992} C_VEL
LIN {X 0,Y 29.623,Z 230.057,A -85,B 0,C 180,E1 -31600.21,E2 -31600.21} C_VEL
LIN {X 0,Y 27.857,Z 217.698,A -85,B 0,C 180,E1 -31612.308,E2 -31612.308} C_VEL
LIN {X 0,Y 27.168,Z 212.06,A -85,B 0,C 180,E1 -31619.539,E2 -31619.539} C_VEL
LIN {X 0,Y 26.093,Z 209.331,A -85,B 0,C 180,E1 -31628.495,E2 -31628.495} C_VEL
LIN {X 0,Y 25.462,Z 206.315,A -85,B 0,C 180,E1 -31646.5,E2 -31646.5} C_VEL
LIN {X 0,Y 25.495,Z 206.562,A -85,B 0,C 180,E1 -31652.292,E2 -31652.292} C_VEL
LIN {X 0,Y 26.221,Z 208.846,A -85,B 0,C 180,E1 -31665.429,E2 -31665.429} C_VEL
LIN {X 0,Y 27.235,Z 214.519,A -85,B 0,C 180,E1 -31676.49,E2 -31676.49} C_VEL
LIN {X 0,Y 27.551,Z 217.949,A -85,B 0,C 180,E1 -31680.381,E2 -31680.381} C_VEL
LIN {X 0,Y 27.317,Z 223.625,A -85,B 0,C 180,E1 -31683.835,E2 -31683.835} C_VEL
LIN {X 0,Y 26.391,Z 229.497,A -85,B 0,C 180,E1 -31685.36,E2 -31685.36} C_VEL
LIN {X 0,Y 22.618,Z 245.813,A -85,B 0,C 180,E1 -31686.496,E2 -31686.496} C_VEL
LIN {X 0,Y 16.121,Z 277.538,A -85,B 0,C 180,E1 -31694.734,E2 -31694.734} C_VEL
LIN {X 0,Y 12.342,Z 289.961,A -85,B 0,C 180,E1 -31702.318,E2 -31702.318} C_VEL
LIN {X 0,Y 8.098,Z 301.562,A -85,B 0,C 180,E1 -31720.618,E2 -31720.618} C_VEL
LIN {X 0,Y 5.957,Z 313.464,A -85,B 0,C 180,E1 -31778.506,E2 -31778.506} C_VEL
LIN {X 0,Y 9.625,Z 322.138,A -85,B 0,C 180,E1 -31816.921,E2 -31816.921} C_VEL
LIN {X 0,Y 8.83,Z 321.137,A -85,B 0,C 180,E1 -31822.774,E2 -31822.774} C_VEL
LIN {X 0,Y 4.038,Z 310.023,A -85,B 0,C 180,E1 -31885.755,E2 -31885.755} C_VEL
LIN {X 0,Y 7.537,Z 298.3,A -85,B 0,C 180,E1 -31944.926,E2 -31944.926} C_VEL
LIN {X 0,Y 12.446,Z 285.622,A -85,B 0,C 180,E1 -31958.942,E2 -31958.942} C_VEL
LIN {X 0,Y 16.498,Z 272.111,A -85,B 0,C 180,E1 -31963.907,E2 -31963.907} C_VEL
LIN {X 0,Y 24.804,Z 231.817,A -85,B 0,C 180,E1 -31971.226,E2 -31971.226} C_VEL
LIN {X 0,Y 24.392,Z 222.201,A -85,B 0,C 180,E1 -31982.187,E2 -31982.187} C_VEL
LIN {X 0,Y 24.37,Z 216.896,A -85,B 0,C 180,E1 -31989.706,E2 -31989.706} C_VEL
LIN {X 0,Y 24.021,Z 215.24,A -85,B 0,C 180,E1 -31997.236,E2 -31997.236} C_VEL
LIN {X 0,Y 24.066,Z 213.401,A -85,B 0,C 180,E1 -32008.456,E2 -32008.456} C_VEL
LIN {X 0,Y 24.14,Z 214.783,A -85,B 0,C 180,E1 -32017.371,E2 -32017.371} C_VEL
LIN {X 0,Y 24.232,Z 219.976,A -85,B 0,C 180,E1 -32027.701,E2 -32027.701} C_VEL
LIN {X 0,Y 24.454,Z 225.868,A -85,B 0,C 180,E1 -32035.64,E2 -32035.64} C_VEL
LIN {X 0,Y 24.355,Z 233.117,A -85,B 0,C 180,E1 -32041.815,E2 -32041.815} C_VEL
LIN {X 0,Y 23.189,Z 242.901,A -85,B 0,C 180,E1 -32045.94,E2 -32045.94} C_VEL
LIN {X 0,Y 22.618,Z 245.813,A -85,B 0,C 180,E1 -32046.496,E2 -32046.496} C_VEL
LIN {X 0,Y 21.104,Z 251.519,A -85,B 0,C 180,E1 -32046.201,E2 -32046.201} C_VEL
LIN {X 0,Y 14.215,Z 269.676,A -85,B 0,C 180,E1 -32032.615,E2 -32032.615} C_VEL
LIN {X 0,Y 12.51,Z 275.319,A -85,B 0,C 180,E1 -32030.591,E2 -32030.591} C_VEL
LIN {X 0,Y 8.909,Z 286.626,A -85,B 0,C 180,E1 -32030.344,E2 -32030.344} C_VEL
LIN {X 0,Y 4.849,Z 296.301,A -85,B 0,C 180,E1 -32026.899,E2 -32026.899} C_VEL
LIN {X 0,Y 4.219,Z 297.101,A -85,B 0,C 180,E1 -32011.164,E2 -32011.164} C_VEL
LIN {X 0,Y 9.118,Z 284.709,A -85,B 0,C 180,E1 -31992.763,E2 -31992.763} C_VEL
LIN {X 0,Y 13.262,Z 270.606,A -85,B 0,C 180,E1 -31988.147,E2 -31988.147} C_VEL
LIN {X 0,Y 21.399,Z 232.738,A -85,B 0,C 180,E1 -31987,E2 -31987} C_VEL
LIN {X 0,Y 22.436,Z 222.224,A -85,B 0,C 180,E1 -32001.217,E2 -32001.217} C_VEL
LIN {X 0,Y 22.49,Z 221.339,A -85,B 0,C 180,E1 -32005.957,E2 -32005.957} C_VEL
LIN {X 0,Y 22.488,Z 221.342,A -85,B 0,C 180,E1 -32009.07,E2 -32009.07} C_VEL
LIN {X 0,Y 21.761,Z 227.159,A -85,B 0,C 180,E1 -32019.117,E2 -32019.117} C_VEL
LIN {X 0,Y 20.975,Z 234.39,A -85,B 0,C 180,E1 -32026.173,E2 -32026.173} C_VEL
LIN {X 0,Y 19.605,Z 242.838,A -85,B 0,C 180,E1 -32029.456,E2 -32029.456} C_VEL
LIN {X 0,Y 12.51,Z 275.319,A -85,B 0,C 180,E1 -32030.591,E2 -32030.591} C_VEL
LIN {X 0,Y 12.44,Z 275.842,A -85,B 0,C 180,E1 -32030.623,E2 -32030.623} C_VEL
LIN {X 0,Y 12.44,Z 600,A -85,B 0,C 180,E1 -32030.623,E2 -32030.623} C_VEL
LIN {X 0,Y 12.44,Z 600,A -85,B 0,C 180,E1 -32030.623,E2 -32030.623}

QRS_NEXT_CUT()

QRS_NEXT()
QRS_HOME()

END
